// TwinCAT 3 PLC project SAsetGains
// ProgramVersion: 3.1.4023.0
// libraries:
//   Tc2_EtherCAT, * (Beckhoff Automation GmbH)
//   Tc2_Standard, * (Beckhoff Automation GmbH)
//   Tc2_System, * (Beckhoff Automation GmbH)
//   Tc3_Module, * (Beckhoff Automation GmbH)
// project tree:
//   / PlcTask.TcTTO
//   POUs/ clear_fault.TcPOU, MAIN.TcPOU, read_alias.TcPOU, read_dongle.TcPOU, read_ncyl.TcPOU, read_write_SA_gains.TcPOU, save_soc.TcPOU, write_gains.TcPOU
// real-time tasks:
//   TASK PlcTask: cycle T#10ms, priority 20, ADS port 350
// motion (NC):
//   TASK NC-Task 1 SAF: cycle T#2ms, priority 4, ADS port 501
//   TASK NC-Task 1 SVB: cycle T#10ms, priority 8, ADS port 511
//   AXIS Axis 1 (id 1)
//     OtherSettings: AllowMotionCmdToSlave=true
//     encoder EncType=19
//       EncPara: MaxCount=#xffffffff
//     drive DrvType=16
//       DrvPara: MaxCount=#xffffffff, DriveControlDWord=#x00020100
//         Analog: TorqueSetpointScale=10, ScaleFactorActTorque=0.1
//         TimeComp: TaskDelayCycles=1
//     controller CtrType=1
//       CtrPara: PriorControlFactor=1
//         Observer: BandWidth=20
//   AXIS Axis 2 (id 2)
//     OtherSettings: AllowMotionCmdToSlave=true
//     encoder EncType=19
//       EncPara: MaxCount=#xffffffff
//     drive DrvType=16
//       DrvPara: MaxCount=#xffffffff, DriveControlDWord=#x00020100
//         Analog: TorqueSetpointScale=10, ScaleFactorActTorque=0.1
//         TimeComp: TaskDelayCycles=1
//     controller CtrType=1
//       CtrPara: PriorControlFactor=1
//         Observer: BandWidth=20
//   AXIS Axis 3 (id 3)
//     OtherSettings: AllowMotionCmdToSlave=true
//     encoder EncType=19
//       EncPara: MaxCount=#xffffffff
//     drive DrvType=16
//       DrvPara: MaxCount=#xffffffff, DriveControlDWord=#x00020100
//         Analog: TorqueSetpointScale=10, ScaleFactorActTorque=0.1
//         TimeComp: TaskDelayCycles=1
//     controller CtrType=1
//       CtrPara: PriorControlFactor=1
//         Observer: BandWidth=20
//   AXIS Axis 4 (id 4)
//     OtherSettings: AllowMotionCmdToSlave=true
//     encoder EncType=19
//       EncPara: MaxCount=#xffffffff
//     drive DrvType=16
//       DrvPara: MaxCount=#xffffffff, DriveControlDWord=#x00020100
//         Analog: TorqueSetpointScale=10, ScaleFactorActTorque=0.1
//         TimeComp: TaskDelayCycles=1
//     controller CtrType=1
//       CtrPara: PriorControlFactor=1
//         Observer: BandWidth=20
//   AXIS Axis 5 (id 5)
//     OtherSettings: AllowMotionCmdToSlave=true
//     encoder EncType=19
//       EncPara: MaxCount=#xffffffff
//     drive DrvType=16
//       DrvPara: MaxCount=#xffffffff, DriveControlDWord=#x00020100
//         Analog: TorqueSetpointScale=10, ScaleFactorActTorque=0.1
//         TimeComp: TaskDelayCycles=1
//     controller CtrType=1
//       CtrPara: PriorControlFactor=1
//         Observer: BandWidth=20
//   AXIS Axis 6 (id 6)
//     OtherSettings: AllowMotionCmdToSlave=true
//     encoder EncType=19
//       EncPara: MaxCount=#xffffffff
//     drive DrvType=16
//       DrvPara: MaxCount=#xffffffff, DriveControlDWord=#x00020100
//         Analog: TorqueSetpointScale=10, ScaleFactorActTorque=0.1
//         TimeComp: TaskDelayCycles=1
//     controller CtrType=1
//       CtrPara: PriorControlFactor=1
//         Observer: BandWidth=20
// I/O:
//   DEVICE Device 1 (EtherCAT), AmsNetId 10.10.16.19.2.1
//     Box 1 (m1eph) [m1eph]
//       Box 2 (m1sa) [m1sa]
//       Box 3 (m1sa) [m1sa]
//       Box 4 (m1sa) [m1sa]
//       Box 5 (m1sa) [m1sa]
//       Box 6 (m1sa) [m1sa]
//       Box 7 (m1sa) [m1sa]
//       Box 8 (m1sa) [m1sa]
//       Box 9 (m1sa) [m1sa]
//       Box 10 (m1sa) [m1sa]
//       Box 11 (m1sa) [m1sa]
//       Box 12 (m1sa) [m1sa]
//       Box 13 (m1sa) [m1sa]
//       Box 14 (m1sa) [m1sa]
//       Box 15 (m1sa) [m1sa]
//       Box 16 (m1sa) [m1sa]
//       Box 17 (m1sa) [m1sa]
//     Box 18 (m1eph) [m1eph]
//       Box 19 (m1sa) [m1sa]
//       Box 20 (m1sa) [m1sa]
//       Box 21 (m1sa) [m1sa]
//       Box 22 (m1sa) [m1sa]
//       Box 23 (m1sa) [m1sa]
//       Box 24 (m1sa) [m1sa]
//       Box 25 (m1sa) [m1sa]
//       Box 26 (m1sa) [m1sa]
//       Box 27 (m1sa) [m1sa]
//       Box 28 (m1sa) [m1sa]
//       Box 29 (m1sa) [m1sa]
//       Box 30 (m1sa) [m1sa]
//       Box 31 (m1sa) [m1sa]
//       Box 32 (m1sa) [m1sa]
//     Box 33 (m1eph) [m1eph]
//       Box 34 (m1sa) [m1sa]
//       Box 35 (m1sa) [m1sa]
//       Box 36 (m1sa) [m1sa]
//       Box 37 (m1sa) [m1sa]
//       Box 38 (m1sa) [m1sa]
//       Box 39 (m1sa) [m1sa]
//       Box 40 (m1sa) [m1sa]
//       Box 41 (m1sa) [m1sa]
//       Box 42 (m1sa) [m1sa]
//       Box 43 (m1sa) [m1sa]
//       Box 44 (m1sa) [m1sa]
//       Box 45 (m1sa) [m1sa]
//     Box 46 (m1eph) [m1eph]
//       Box 47 (m1sa) [m1sa]
//       Box 48 (m1sa) [m1sa]
//       Box 49 (m1sa) [m1sa]
//       Box 50 (m1sa) [m1sa]
//       Box 51 (m1sa) [m1sa]
//       Box 52 (m1sa) [m1sa]
//       Box 53 (m1sa) [m1sa]
//       Box 54 (m1sa) [m1sa]
//       Box 55 (m1sa) [m1sa]
//       Box 56 (m1sa) [m1sa]
//       Box 57 (m1sa) [m1sa]
//       Box 58 (m1sa) [m1sa]
//       Box 59 (m1sa) [m1sa]
//       Box 60 (m1sa) [m1sa]
//       Box 61 (m1sa) [m1sa]
//       Box 62 (m1sa) [m1sa]
//     Box 63 (m1eph) [m1eph]
//       Box 64 (m1sa) [m1sa]
//       Box 65 (m1sa) [m1sa]
//       Box 66 (m1sa) [m1sa]
//       Box 67 (m1sa) [m1sa]
//       Box 68 (m1sa) [m1sa]
//       Box 69 (m1sa) [m1sa]
//       Box 70 (m1sa) [m1sa]
//       Box 71 (m1sa) [m1sa]
//       Box 72 (m1sa) [m1sa]
//       Box 73 (m1sa) [m1sa]
//       Box 74 (m1sa) [m1sa]
//       Box 75 (m1sa) [m1sa]
//       Box 76 (m1sa) [m1sa]
//       Box 77 (m1sa) [m1sa]
//       Box 78 (m1sa) [m1sa]
//       Box 79 (m1sa) [m1sa]
//     Box 80 (m1eph) [m1eph]
//       Box 81 (m1sa) [m1sa]
//       Box 82 (m1sa) [m1sa]
//       Box 83 (m1sa) [m1sa]
//       Box 84 (m1sa) [m1sa]
//       Box 85 (m1sa) [m1sa]
//       Box 86 (m1sa) [m1sa]
//       Box 87 (m1sa) [m1sa]
//       Box 88 (m1sa) [m1sa]
//       Box 89 (m1sa) [m1sa]
//       Box 90 (m1sa) [m1sa]
//       Box 91 (m1sa) [m1sa]
//       Box 92 (m1sa) [m1sa]
//       Box 93 (m1sa) [m1sa]
//       Box 94 (m1sa) [m1sa]
//       Box 95 (m1sa) [m1sa]
//       Box 96 (m1sa) [m1sa]
//     Box 97 (m1eph) [m1eph]
//       Box 98 (m1sa) [m1sa]
//       Box 99 (m1sa) [m1sa]
//       Box 100 (m1sa) [m1sa]
//       Box 101 (m1sa) [m1sa]
//       Box 102 (m1sa) [m1sa]
//       Box 103 (m1sa) [m1sa]
//       Box 104 (m1sa) [m1sa]
//       Box 105 (m1sa) [m1sa]
//       Box 106 (m1sa) [m1sa]
//       Box 107 (m1sa) [m1sa]
//       Box 108 (m1sa) [m1sa]
//       Box 109 (m1sa) [m1sa]
//       Box 110 (m1sa) [m1sa]
//       Box 111 (m1sa) [m1sa]
//       Box 112 (m1sa) [m1sa]
//       Box 113 (m1sa) [m1sa]
//     Box 114 (m1eph) [m1eph]
//       Box 115 (m1sa) [m1sa]
//       Box 116 (m1sa) [m1sa]
//       Box 117 (m1sa) [m1sa]
//       Box 118 (m1sa) [m1sa]
//       Box 119 (m1sa) [m1sa]
//       Box 120 (m1sa) [m1sa]
//       Box 121 (m1sa) [m1sa]
//       Box 122 (m1sa) [m1sa]
//       Box 123 (m1sa) [m1sa]
//       Box 124 (m1sa) [m1sa]
//       Box 125 (m1sa) [m1sa]
//       Box 126 (m1sa) [m1sa]
//       Box 127 (m1sa) [m1sa]
//       Box 128 (m1sa) [m1sa]
//       Box 129 (m1sa) [m1sa]
//       Box 130 (m1sa) [m1sa]
//     Box 131 (m1eph) [m1eph]
//       Box 132 (m1sa) [m1sa]
//       Box 133 (m1sa) [m1sa]
//       Box 134 (m1sa) [m1sa]
//       Box 135 (m1sa) [m1sa]
//       Box 136 (m1sa) [m1sa]
//       Box 137 (m1sa) [m1sa]
//       Box 138 (m1sa) [m1sa]
//       Box 139 (m1sa) [m1sa]
//       Box 140 (m1sa) [m1sa]
//       Box 141 (m1sa) [m1sa]
//       Box 142 (m1sa) [m1sa]
//       Box 143 (m1sa) [m1sa]
//       Box 144 (m1sa) [m1sa]
//       Box 145 (m1sa) [m1sa]
//       Box 146 (m1sa) [m1sa]
//       Box 147 (m1sa) [m1sa]
//     Box 148 (m1eph) [m1eph]
//       Box 149 (m1sa) [m1sa]
//       Box 150 (m1sa) [m1sa]
//       Box 151 (m1sa) [m1sa]
//       Box 152 (m1sa) [m1sa]
//       Box 153 (m1sa) [m1sa]
//       Box 154 (m1sa) [m1sa]
//       Box 155 (m1sa) [m1sa]
//       Box 156 (m1sa) [m1sa]
//       Box 157 (m1sa) [m1sa]
//       Box 158 (m1sa) [m1sa]
//       Box 159 (m1sa) [m1sa]
//       Box 160 (m1sa) [m1sa]
//       Box 161 (m1sa) [m1sa]
//       Box 162 (m1sa) [m1sa]
//       Box 163 (m1sa) [m1sa]
//       Box 164 (m1sa) [m1sa]
//     Box 165 (m1eph) [m1eph]
//       Box 166 (m1sa) [m1sa]
//       Box 167 (m1sa) [m1sa]
//       Box 168 (m1sa) [m1sa]
//       Box 169 (m1sa) [m1sa]
//       Box 170 (m1sa) [m1sa]
//       Box 171 (m1sa) [m1sa]
//       Box 172 (m1sa) [m1sa]
//       Box 173 (m1sa) [m1sa]
//       Box 174 (m1sa) [m1sa]
//       Box 175 (m1sa) [m1sa]
//       Box 176 (m1sa) [m1sa]
//       Box 177 (m1sa) [m1sa]
//       Box 178 (m1sa) [m1sa]
//       Box 179 (m1sa) [m1sa]
//       Box 180 (m1sa) [m1sa]
//       Box 181 (m1sa) [m1sa]
//     Drive 182 (BEL) [BEL]
//       modules: Module 1 (Cyclic position Mode)
//     Term 183 (EK1100) [EK1100 EtherCAT Coupler (2A E-Bus)]
//       Term 184 (EL5042) [EL5042 2Ch. BiSS-C Encoder]
//       Term 185 (EL3312) [EL3312 2Ch. Ana. Input Thermocouple (TC)]
//       Term 186 (EL9505) [EL9505 Power supply terminal 5V]
//       Term 187 (EL3356-0010) [EL3356-0010 1Ch. Ana. Input Resistor Bridge Terminal, 24bit, High Precision]
//       Term 218 (EL9011) [EL9011 End Terminal]
//     Drive 188 (BEL) [BEL]
//       modules: Module 1 (Cyclic position Mode)
//     Term 189 (EK1100) [EK1100 EtherCAT Coupler (2A E-Bus)]
//       Term 190 (EL5042) [EL5042 2Ch. BiSS-C Encoder]
//       Term 191 (EL3312) [EL3312 2Ch. Ana. Input Thermocouple (TC)]
//       Term 192 (EL9505) [EL9505 Power supply terminal 5V]
//       Term 193 (EL3356-0010) [EL3356-0010 1Ch. Ana. Input Resistor Bridge Terminal, 24bit, High Precision]
//       Term 219 (EL9011) [EL9011 End Terminal]
//     Drive 194 (BEL) [BEL]
//       modules: Module 1 (Cyclic position Mode)
//     Term 195 (EK1100) [EK1100 EtherCAT Coupler (2A E-Bus)]
//       Term 196 (EL5042) [EL5042 2Ch. BiSS-C Encoder]
//       Term 197 (EL3312) [EL3312 2Ch. Ana. Input Thermocouple (TC)]
//       Term 198 (EL9505) [EL9505 Power supply terminal 5V]
//       Term 199 (EL3356-0010) [EL3356-0010 1Ch. Ana. Input Resistor Bridge Terminal, 24bit, High Precision]
//       Term 220 (EL9011) [EL9011 End Terminal]
//     Drive 200 (BEL) [BEL]
//       modules: Module 1 (Cyclic position Mode)
//     Term 201 (EK1100) [EK1100 EtherCAT Coupler (2A E-Bus)]
//       Term 202 (EL5042) [EL5042 2Ch. BiSS-C Encoder]
//       Term 203 (EL3312) [EL3312 2Ch. Ana. Input Thermocouple (TC)]
//       Term 204 (EL9505) [EL9505 Power supply terminal 5V]
//       Term 205 (EL3356-0010) [EL3356-0010 1Ch. Ana. Input Resistor Bridge Terminal, 24bit, High Precision]
//       Term 221 (EL9011) [EL9011 End Terminal]
//     Drive 206 (BEL) [BEL]
//       modules: Module 1 (Cyclic position Mode)
//     Term 207 (EK1100) [EK1100 EtherCAT Coupler (2A E-Bus)]
//       Term 208 (EL5042) [EL5042 2Ch. BiSS-C Encoder]
//       Term 209 (EL3312) [EL3312 2Ch. Ana. Input Thermocouple (TC)]
//       Term 210 (EL9505) [EL9505 Power supply terminal 5V]
//       Term 211 (EL3356-0010) [EL3356-0010 1Ch. Ana. Input Resistor Bridge Terminal, 24bit, High Precision]
//       Term 222 (EL9011) [EL9011 End Terminal]
//     Drive 212 (BEL) [BEL]
//       modules: Module 1 (Cyclic position Mode)
//     Term 213 (EK1100) [EK1100 EtherCAT Coupler (2A E-Bus)]
//       Term 214 (EL5042) [EL5042 2Ch. BiSS-C Encoder]
//       Term 215 (EL3312) [EL3312 2Ch. Ana. Input Thermocouple (TC)]
//       Term 216 (EL9505) [EL9505 Power supply terminal 5V]
//       Term 217 (EL3356-0010) [EL3356-0010 1Ch. Ana. Input Resistor Bridge Terminal, 24bit, High Precision]
//       Term 223 (EL9011) [EL9011 End Terminal]
// variable links:
//   NC-Task 1 SAF/Axes/Axis 1 <-> Device 1 (EtherCAT)/Drive 182 (BEL)
//     Drive/Inputs/In/nDataIn1 <-> Module 1 (Cyclic position Mode)/Cyclic position Inputs/Position loop error
//     Drive/Inputs/In/nDataIn3[0] <-> Module 1 (Cyclic position Mode)/Cyclic position Inputs/Torque actual value
//     Drive/Inputs/In/nDcOutputTime <-> InfoData/DcOutputShift
//     Drive/Inputs/In/nState1 <-> Module 1 (Cyclic position Mode)/Cyclic position Inputs/Status word
//     Drive/Inputs/In/nState2 <-> Module 1 (Cyclic position Mode)/Cyclic position Inputs/Status word @bit 8
//     Drive/Inputs/In/nState4 @bit 1 <-> WcState/InputToggle
//     Drive/Inputs/In/nState4 <-> WcState/WcState
//     Drive/Outputs/Out/nCtrl1 <-> Module 1 (Cyclic position Mode)/Cyclic position Outputs/Control word
//     Drive/Outputs/Out/nCtrl2 <-> Module 1 (Cyclic position Mode)/Cyclic position Outputs/Control word @bit 8
//     Drive/Outputs/Out/nDataOut1 <-> Module 1 (Cyclic position Mode)/Cyclic position Outputs/Profile target position
//     Drive/Outputs/Out/nDataOut3[0] <-> Module 1 (Cyclic position Mode)/Cyclic position Outputs/Torque offset
//     Enc/Inputs/In/nDataIn1 <-> Module 1 (Cyclic position Mode)/Cyclic position Inputs/Actual motor position
//     Enc/Inputs/In/nDataIn7 <-> Module 1 (Cyclic position Mode)/Cyclic position Inputs/Actual motor velocity
//     Enc/Inputs/In/nDcInputTime <-> InfoData/DcInputShift
//     Enc/Inputs/In/nState4 @bit 1 <-> WcState/InputToggle
//     Enc/Inputs/In/nState4 <-> WcState/WcState
//   NC-Task 1 SAF/Axes/Axis 2 <-> Device 1 (EtherCAT)/Drive 188 (BEL)
//     Drive/Inputs/In/nDataIn1 <-> Module 1 (Cyclic position Mode)/Cyclic position Inputs/Position loop error
//     Drive/Inputs/In/nDataIn3[0] <-> Module 1 (Cyclic position Mode)/Cyclic position Inputs/Torque actual value
//     Drive/Inputs/In/nDcOutputTime <-> InfoData/DcOutputShift
//     Drive/Inputs/In/nState1 <-> Module 1 (Cyclic position Mode)/Cyclic position Inputs/Status word
//     Drive/Inputs/In/nState2 <-> Module 1 (Cyclic position Mode)/Cyclic position Inputs/Status word @bit 8
//     Drive/Inputs/In/nState4 @bit 1 <-> WcState/InputToggle
//     Drive/Inputs/In/nState4 <-> WcState/WcState
//     Drive/Outputs/Out/nCtrl1 <-> Module 1 (Cyclic position Mode)/Cyclic position Outputs/Control word
//     Drive/Outputs/Out/nCtrl2 <-> Module 1 (Cyclic position Mode)/Cyclic position Outputs/Control word @bit 8
//     Drive/Outputs/Out/nDataOut1 <-> Module 1 (Cyclic position Mode)/Cyclic position Outputs/Profile target position
//     Drive/Outputs/Out/nDataOut3[0] <-> Module 1 (Cyclic position Mode)/Cyclic position Outputs/Torque offset
//     Enc/Inputs/In/nDataIn1 <-> Module 1 (Cyclic position Mode)/Cyclic position Inputs/Actual motor position
//     Enc/Inputs/In/nDataIn7 <-> Module 1 (Cyclic position Mode)/Cyclic position Inputs/Actual motor velocity
//     Enc/Inputs/In/nDcInputTime <-> InfoData/DcInputShift
//     Enc/Inputs/In/nState4 @bit 1 <-> WcState/InputToggle
//     Enc/Inputs/In/nState4 <-> WcState/WcState
//   NC-Task 1 SAF/Axes/Axis 3 <-> Device 1 (EtherCAT)/Drive 194 (BEL)
//     Drive/Inputs/In/nDataIn1 <-> Module 1 (Cyclic position Mode)/Cyclic position Inputs/Position loop error
//     Drive/Inputs/In/nDataIn3[0] <-> Module 1 (Cyclic position Mode)/Cyclic position Inputs/Torque actual value
//     Drive/Inputs/In/nDcOutputTime <-> InfoData/DcOutputShift
//     Drive/Inputs/In/nState1 <-> Module 1 (Cyclic position Mode)/Cyclic position Inputs/Status word
//     Drive/Inputs/In/nState2 <-> Module 1 (Cyclic position Mode)/Cyclic position Inputs/Status word @bit 8
//     Drive/Inputs/In/nState4 @bit 1 <-> WcState/InputToggle
//     Drive/Inputs/In/nState4 <-> WcState/WcState
//     Drive/Outputs/Out/nCtrl1 <-> Module 1 (Cyclic position Mode)/Cyclic position Outputs/Control word
//     Drive/Outputs/Out/nCtrl2 <-> Module 1 (Cyclic position Mode)/Cyclic position Outputs/Control word @bit 8
//     Drive/Outputs/Out/nDataOut1 <-> Module 1 (Cyclic position Mode)/Cyclic position Outputs/Profile target position
//     Drive/Outputs/Out/nDataOut3[0] <-> Module 1 (Cyclic position Mode)/Cyclic position Outputs/Torque offset
//     Enc/Inputs/In/nDataIn1 <-> Module 1 (Cyclic position Mode)/Cyclic position Inputs/Actual motor position
//     Enc/Inputs/In/nDataIn7 <-> Module 1 (Cyclic position Mode)/Cyclic position Inputs/Actual motor velocity
//     Enc/Inputs/In/nDcInputTime <-> InfoData/DcInputShift
//     Enc/Inputs/In/nState4 @bit 1 <-> WcState/InputToggle
//     Enc/Inputs/In/nState4 <-> WcState/WcState
//   NC-Task 1 SAF/Axes/Axis 4 <-> Device 1 (EtherCAT)/Drive 200 (BEL)
//     Drive/Inputs/In/nDataIn1 <-> Module 1 (Cyclic position Mode)/Cyclic position Inputs/Position loop error
//     Drive/Inputs/In/nDataIn3[0] <-> Module 1 (Cyclic position Mode)/Cyclic position Inputs/Torque actual value
//     Drive/Inputs/In/nDcOutputTime <-> InfoData/DcOutputShift
//     Drive/Inputs/In/nState1 <-> Module 1 (Cyclic position Mode)/Cyclic position Inputs/Status word
//     Drive/Inputs/In/nState2 <-> Module 1 (Cyclic position Mode)/Cyclic position Inputs/Status word @bit 8
//     Drive/Inputs/In/nState4 @bit 1 <-> WcState/InputToggle
//     Drive/Inputs/In/nState4 <-> WcState/WcState
//     Drive/Outputs/Out/nCtrl1 <-> Module 1 (Cyclic position Mode)/Cyclic position Outputs/Control word
//     Drive/Outputs/Out/nCtrl2 <-> Module 1 (Cyclic position Mode)/Cyclic position Outputs/Control word @bit 8
//     Drive/Outputs/Out/nDataOut1 <-> Module 1 (Cyclic position Mode)/Cyclic position Outputs/Profile target position
//     Drive/Outputs/Out/nDataOut3[0] <-> Module 1 (Cyclic position Mode)/Cyclic position Outputs/Torque offset
//     Enc/Inputs/In/nDataIn1 <-> Module 1 (Cyclic position Mode)/Cyclic position Inputs/Actual motor position
//     Enc/Inputs/In/nDataIn7 <-> Module 1 (Cyclic position Mode)/Cyclic position Inputs/Actual motor velocity
//     Enc/Inputs/In/nDcInputTime <-> InfoData/DcInputShift
//     Enc/Inputs/In/nState4 @bit 1 <-> WcState/InputToggle
//     Enc/Inputs/In/nState4 <-> WcState/WcState
//   NC-Task 1 SAF/Axes/Axis 5 <-> Device 1 (EtherCAT)/Drive 206 (BEL)
//     Drive/Inputs/In/nDataIn1 <-> Module 1 (Cyclic position Mode)/Cyclic position Inputs/Position loop error
//     Drive/Inputs/In/nDataIn3[0] <-> Module 1 (Cyclic position Mode)/Cyclic position Inputs/Torque actual value
//     Drive/Inputs/In/nDcOutputTime <-> InfoData/DcOutputShift
//     Drive/Inputs/In/nState1 <-> Module 1 (Cyclic position Mode)/Cyclic position Inputs/Status word
//     Drive/Inputs/In/nState2 <-> Module 1 (Cyclic position Mode)/Cyclic position Inputs/Status word @bit 8
//     Drive/Inputs/In/nState4 @bit 1 <-> WcState/InputToggle
//     Drive/Inputs/In/nState4 <-> WcState/WcState
//     Drive/Outputs/Out/nCtrl1 <-> Module 1 (Cyclic position Mode)/Cyclic position Outputs/Control word
//     Drive/Outputs/Out/nCtrl2 <-> Module 1 (Cyclic position Mode)/Cyclic position Outputs/Control word @bit 8
//     Drive/Outputs/Out/nDataOut1 <-> Module 1 (Cyclic position Mode)/Cyclic position Outputs/Profile target position
//     Drive/Outputs/Out/nDataOut3[0] <-> Module 1 (Cyclic position Mode)/Cyclic position Outputs/Torque offset
//     Enc/Inputs/In/nDataIn1 <-> Module 1 (Cyclic position Mode)/Cyclic position Inputs/Actual motor position
//     Enc/Inputs/In/nDataIn7 <-> Module 1 (Cyclic position Mode)/Cyclic position Inputs/Actual motor velocity
//     Enc/Inputs/In/nDcInputTime <-> InfoData/DcInputShift
//     Enc/Inputs/In/nState4 @bit 1 <-> WcState/InputToggle
//     Enc/Inputs/In/nState4 <-> WcState/WcState
//   NC-Task 1 SAF/Axes/Axis 6 <-> Device 1 (EtherCAT)/Drive 212 (BEL)
//     Drive/Inputs/In/nDataIn1 <-> Module 1 (Cyclic position Mode)/Cyclic position Inputs/Position loop error
//     Drive/Inputs/In/nDataIn3[0] <-> Module 1 (Cyclic position Mode)/Cyclic position Inputs/Torque actual value
//     Drive/Inputs/In/nDcOutputTime <-> InfoData/DcOutputShift
//     Drive/Inputs/In/nState1 <-> Module 1 (Cyclic position Mode)/Cyclic position Inputs/Status word
//     Drive/Inputs/In/nState2 <-> Module 1 (Cyclic position Mode)/Cyclic position Inputs/Status word @bit 8
//     Drive/Inputs/In/nState4 @bit 1 <-> WcState/InputToggle
//     Drive/Inputs/In/nState4 <-> WcState/WcState
//     Drive/Outputs/Out/nCtrl1 <-> Module 1 (Cyclic position Mode)/Cyclic position Outputs/Control word
//     Drive/Outputs/Out/nCtrl2 <-> Module 1 (Cyclic position Mode)/Cyclic position Outputs/Control word @bit 8
//     Drive/Outputs/Out/nDataOut1 <-> Module 1 (Cyclic position Mode)/Cyclic position Outputs/Profile target position
//     Drive/Outputs/Out/nDataOut3[0] <-> Module 1 (Cyclic position Mode)/Cyclic position Outputs/Torque offset
//     Enc/Inputs/In/nDataIn1 <-> Module 1 (Cyclic position Mode)/Cyclic position Inputs/Actual motor position
//     Enc/Inputs/In/nDataIn7 <-> Module 1 (Cyclic position Mode)/Cyclic position Inputs/Actual motor velocity
//     Enc/Inputs/In/nDcInputTime <-> InfoData/DcInputShift
//     Enc/Inputs/In/nState4 @bit 1 <-> WcState/InputToggle
//     Enc/Inputs/In/nState4 <-> WcState/WcState
//   SAsetGains/SAsetGains Instance <-> Device 1 (EtherCAT)
//     PlcTask Inputs/MAIN.FrmWcStat[1] <-> Inputs/Frm0WcState
//   SAsetGains/SAsetGains Instance <-> Device 1 (EtherCAT)/Box 1 (m1eph)
//     PlcTask Outputs/MAIN.msthb[1] <-> Control process data mapping/msthb
//   SAsetGains/SAsetGains Instance <-> Device 1 (EtherCAT)/Box 1 (m1eph)/Box 10 (m1sa)
//     PlcTask Inputs/MAIN.cloop_stat[9] <-> Status process data mapping/close_loop
//     PlcTask Inputs/MAIN.enable_stat[9] <-> Status process data mapping/enable
//     PlcTask Inputs/MAIN.force_rb_X[9] <-> Status process data mapping/force_rb_X
//     PlcTask Inputs/MAIN.force_rb_Y[9] <-> Status process data mapping/force_rb_Y
//     PlcTask Inputs/MAIN.force_rb_Z[9] <-> Status process data mapping/force_rb_Z
//     PlcTask Inputs/MAIN.force_sp_X[9] <-> Status process data mapping/force_sp_X
//     PlcTask Inputs/MAIN.force_sp_Y[9] <-> Status process data mapping/force_sp_Y
//     PlcTask Inputs/MAIN.force_sp_Z[9] <-> Status process data mapping/force_sp_Z
//     PlcTask Inputs/MAIN.pwm1[9] <-> Status process data mapping/pwm1
//     PlcTask Inputs/MAIN.pwm2[9] <-> Status process data mapping/pwm2
//     PlcTask Inputs/MAIN.pwm3[9] <-> Status process data mapping/pwm3
//     PlcTask Outputs/MAIN.enable_cmd[9] <-> Control process data mapping/enable
//     PlcTask Outputs/MAIN.force_cmd_X[9] <-> Control process data mapping/force_sp_X
//     PlcTask Outputs/MAIN.force_cmd_Y[9] <-> Control process data mapping/force_sp_Y
//     PlcTask Outputs/MAIN.force_cmd_Z[9] <-> Control process data mapping/force_sp_Z
//     PlcTask Outputs/MAIN.msthb[10] <-> Control process data mapping/msthb
//   SAsetGains/SAsetGains Instance <-> Device 1 (EtherCAT)/Box 1 (m1eph)/Box 11 (m1sa)
//     PlcTask Inputs/MAIN.cloop_stat[10] <-> Status process data mapping/close_loop
//     PlcTask Inputs/MAIN.enable_stat[10] <-> Status process data mapping/enable
//     PlcTask Inputs/MAIN.force_rb_X[10] <-> Status process data mapping/force_rb_X
//     PlcTask Inputs/MAIN.force_rb_Y[10] <-> Status process data mapping/force_rb_Y
//     PlcTask Inputs/MAIN.force_rb_Z[10] <-> Status process data mapping/force_rb_Z
//     PlcTask Inputs/MAIN.force_sp_X[10] <-> Status process data mapping/force_sp_X
//     PlcTask Inputs/MAIN.force_sp_Y[10] <-> Status process data mapping/force_sp_Y
//     PlcTask Inputs/MAIN.force_sp_Z[10] <-> Status process data mapping/force_sp_Z
//     PlcTask Inputs/MAIN.pwm1[10] <-> Status process data mapping/pwm1
//     PlcTask Inputs/MAIN.pwm2[10] <-> Status process data mapping/pwm2
//     PlcTask Inputs/MAIN.pwm3[10] <-> Status process data mapping/pwm3
//     PlcTask Outputs/MAIN.enable_cmd[10] <-> Control process data mapping/enable
//     PlcTask Outputs/MAIN.force_cmd_X[10] <-> Control process data mapping/force_sp_X
//     PlcTask Outputs/MAIN.force_cmd_Y[10] <-> Control process data mapping/force_sp_Y
//     PlcTask Outputs/MAIN.force_cmd_Z[10] <-> Control process data mapping/force_sp_Z
//     PlcTask Outputs/MAIN.msthb[11] <-> Control process data mapping/msthb
//   SAsetGains/SAsetGains Instance <-> Device 1 (EtherCAT)/Box 1 (m1eph)/Box 12 (m1sa)
//     PlcTask Inputs/MAIN.cloop_stat[11] <-> Status process data mapping/close_loop
//     PlcTask Inputs/MAIN.enable_stat[11] <-> Status process data mapping/enable
//     PlcTask Inputs/MAIN.force_rb_X[11] <-> Status process data mapping/force_rb_X
//     PlcTask Inputs/MAIN.force_rb_Y[11] <-> Status process data mapping/force_rb_Y
//     PlcTask Inputs/MAIN.force_rb_Z[11] <-> Status process data mapping/force_rb_Z
//     PlcTask Inputs/MAIN.force_sp_X[11] <-> Status process data mapping/force_sp_X
//     PlcTask Inputs/MAIN.force_sp_Y[11] <-> Status process data mapping/force_sp_Y
//     PlcTask Inputs/MAIN.force_sp_Z[11] <-> Status process data mapping/force_sp_Z
//     PlcTask Inputs/MAIN.pwm1[11] <-> Status process data mapping/pwm1
//     PlcTask Inputs/MAIN.pwm2[11] <-> Status process data mapping/pwm2
//     PlcTask Inputs/MAIN.pwm3[11] <-> Status process data mapping/pwm3
//     PlcTask Outputs/MAIN.enable_cmd[11] <-> Control process data mapping/enable
//     PlcTask Outputs/MAIN.force_cmd_X[11] <-> Control process data mapping/force_sp_X
//     PlcTask Outputs/MAIN.force_cmd_Y[11] <-> Control process data mapping/force_sp_Y
//     PlcTask Outputs/MAIN.force_cmd_Z[11] <-> Control process data mapping/force_sp_Z
//     PlcTask Outputs/MAIN.msthb[12] <-> Control process data mapping/msthb
//   SAsetGains/SAsetGains Instance <-> Device 1 (EtherCAT)/Box 1 (m1eph)/Box 13 (m1sa)
//     PlcTask Inputs/MAIN.cloop_stat[12] <-> Status process data mapping/close_loop
//     PlcTask Inputs/MAIN.enable_stat[12] <-> Status process data mapping/enable
//     PlcTask Inputs/MAIN.force_rb_X[12] <-> Status process data mapping/force_rb_X
//     PlcTask Inputs/MAIN.force_rb_Y[12] <-> Status process data mapping/force_rb_Y
//     PlcTask Inputs/MAIN.force_rb_Z[12] <-> Status process data mapping/force_rb_Z
//     PlcTask Inputs/MAIN.force_sp_X[12] <-> Status process data mapping/force_sp_X
//     PlcTask Inputs/MAIN.force_sp_Y[12] <-> Status process data mapping/force_sp_Y
//     PlcTask Inputs/MAIN.force_sp_Z[12] <-> Status process data mapping/force_sp_Z
//     PlcTask Inputs/MAIN.pwm1[12] <-> Status process data mapping/pwm1
//     PlcTask Inputs/MAIN.pwm2[12] <-> Status process data mapping/pwm2
//     PlcTask Inputs/MAIN.pwm3[12] <-> Status process data mapping/pwm3
//     PlcTask Outputs/MAIN.enable_cmd[12] <-> Control process data mapping/enable
//     PlcTask Outputs/MAIN.force_cmd_X[12] <-> Control process data mapping/force_sp_X
//     PlcTask Outputs/MAIN.force_cmd_Y[12] <-> Control process data mapping/force_sp_Y
//     PlcTask Outputs/MAIN.force_cmd_Z[12] <-> Control process data mapping/force_sp_Z
//     PlcTask Outputs/MAIN.msthb[13] <-> Control process data mapping/msthb
//   SAsetGains/SAsetGains Instance <-> Device 1 (EtherCAT)/Box 1 (m1eph)/Box 14 (m1sa)
//     PlcTask Inputs/MAIN.cloop_stat[13] <-> Status process data mapping/close_loop
//     PlcTask Inputs/MAIN.enable_stat[13] <-> Status process data mapping/enable
//     PlcTask Inputs/MAIN.force_rb_X[13] <-> Status process data mapping/force_rb_X
//     PlcTask Inputs/MAIN.force_rb_Y[13] <-> Status process data mapping/force_rb_Y
//     PlcTask Inputs/MAIN.force_rb_Z[13] <-> Status process data mapping/force_rb_Z
//     PlcTask Inputs/MAIN.force_sp_X[13] <-> Status process data mapping/force_sp_X
//     PlcTask Inputs/MAIN.force_sp_Y[13] <-> Status process data mapping/force_sp_Y
//     PlcTask Inputs/MAIN.force_sp_Z[13] <-> Status process data mapping/force_sp_Z
//     PlcTask Inputs/MAIN.pwm1[13] <-> Status process data mapping/pwm1
//     PlcTask Inputs/MAIN.pwm2[13] <-> Status process data mapping/pwm2
//     PlcTask Inputs/MAIN.pwm3[13] <-> Status process data mapping/pwm3
//     PlcTask Outputs/MAIN.enable_cmd[13] <-> Control process data mapping/enable
//     PlcTask Outputs/MAIN.force_cmd_X[13] <-> Control process data mapping/force_sp_X
//     PlcTask Outputs/MAIN.force_cmd_Y[13] <-> Control process data mapping/force_sp_Y
//     PlcTask Outputs/MAIN.force_cmd_Z[13] <-> Control process data mapping/force_sp_Z
//     PlcTask Outputs/MAIN.msthb[14] <-> Control process data mapping/msthb
//   SAsetGains/SAsetGains Instance <-> Device 1 (EtherCAT)/Box 1 (m1eph)/Box 15 (m1sa)
//     PlcTask Inputs/MAIN.cloop_stat[14] <-> Status process data mapping/close_loop
//     PlcTask Inputs/MAIN.enable_stat[14] <-> Status process data mapping/enable
//     PlcTask Inputs/MAIN.force_rb_X[14] <-> Status process data mapping/force_rb_X
//     PlcTask Inputs/MAIN.force_rb_Y[14] <-> Status process data mapping/force_rb_Y
//     PlcTask Inputs/MAIN.force_rb_Z[14] <-> Status process data mapping/force_rb_Z
//     PlcTask Inputs/MAIN.force_sp_X[14] <-> Status process data mapping/force_sp_X
//     PlcTask Inputs/MAIN.force_sp_Y[14] <-> Status process data mapping/force_sp_Y
//     PlcTask Inputs/MAIN.force_sp_Z[14] <-> Status process data mapping/force_sp_Z
//     PlcTask Inputs/MAIN.pwm1[14] <-> Status process data mapping/pwm1
//     PlcTask Inputs/MAIN.pwm2[14] <-> Status process data mapping/pwm2
//     PlcTask Inputs/MAIN.pwm3[14] <-> Status process data mapping/pwm3
//     PlcTask Outputs/MAIN.enable_cmd[14] <-> Control process data mapping/enable
//     PlcTask Outputs/MAIN.force_cmd_X[14] <-> Control process data mapping/force_sp_X
//     PlcTask Outputs/MAIN.force_cmd_Y[14] <-> Control process data mapping/force_sp_Y
//     PlcTask Outputs/MAIN.force_cmd_Z[14] <-> Control process data mapping/force_sp_Z
//     PlcTask Outputs/MAIN.msthb[15] <-> Control process data mapping/msthb
//   SAsetGains/SAsetGains Instance <-> Device 1 (EtherCAT)/Box 1 (m1eph)/Box 16 (m1sa)
//     PlcTask Inputs/MAIN.cloop_stat[15] <-> Status process data mapping/close_loop
//     PlcTask Inputs/MAIN.enable_stat[15] <-> Status process data mapping/enable
//     PlcTask Inputs/MAIN.force_rb_X[15] <-> Status process data mapping/force_rb_X
//     PlcTask Inputs/MAIN.force_rb_Y[15] <-> Status process data mapping/force_rb_Y
//     PlcTask Inputs/MAIN.force_rb_Z[15] <-> Status process data mapping/force_rb_Z
//     PlcTask Inputs/MAIN.force_sp_X[15] <-> Status process data mapping/force_sp_X
//     PlcTask Inputs/MAIN.force_sp_Y[15] <-> Status process data mapping/force_sp_Y
//     PlcTask Inputs/MAIN.force_sp_Z[15] <-> Status process data mapping/force_sp_Z
//     PlcTask Inputs/MAIN.pwm1[15] <-> Status process data mapping/pwm1
//     PlcTask Inputs/MAIN.pwm2[15] <-> Status process data mapping/pwm2
//     PlcTask Inputs/MAIN.pwm3[15] <-> Status process data mapping/pwm3
//     PlcTask Outputs/MAIN.enable_cmd[15] <-> Control process data mapping/enable
//     PlcTask Outputs/MAIN.force_cmd_X[15] <-> Control process data mapping/force_sp_X
//     PlcTask Outputs/MAIN.force_cmd_Y[15] <-> Control process data mapping/force_sp_Y
//     PlcTask Outputs/MAIN.force_cmd_Z[15] <-> Control process data mapping/force_sp_Z
//     PlcTask Outputs/MAIN.msthb[16] <-> Control process data mapping/msthb
//   SAsetGains/SAsetGains Instance <-> Device 1 (EtherCAT)/Box 1 (m1eph)/Box 17 (m1sa)
//     PlcTask Inputs/MAIN.cloop_stat[16] <-> Status process data mapping/close_loop
//     PlcTask Inputs/MAIN.enable_stat[16] <-> Status process data mapping/enable
//     PlcTask Inputs/MAIN.force_rb_X[16] <-> Status process data mapping/force_rb_X
//     PlcTask Inputs/MAIN.force_rb_Y[16] <-> Status process data mapping/force_rb_Y
//     PlcTask Inputs/MAIN.force_rb_Z[16] <-> Status process data mapping/force_rb_Z
//     PlcTask Inputs/MAIN.force_sp_X[16] <-> Status process data mapping/force_sp_X
//     PlcTask Inputs/MAIN.force_sp_Y[16] <-> Status process data mapping/force_sp_Y
//     PlcTask Inputs/MAIN.force_sp_Z[16] <-> Status process data mapping/force_sp_Z
//     PlcTask Inputs/MAIN.pwm1[16] <-> Status process data mapping/pwm1
//     PlcTask Inputs/MAIN.pwm2[16] <-> Status process data mapping/pwm2
//     PlcTask Inputs/MAIN.pwm3[16] <-> Status process data mapping/pwm3
//     PlcTask Outputs/MAIN.enable_cmd[16] <-> Control process data mapping/enable
//     PlcTask Outputs/MAIN.force_cmd_X[16] <-> Control process data mapping/force_sp_X
//     PlcTask Outputs/MAIN.force_cmd_Y[16] <-> Control process data mapping/force_sp_Y
//     PlcTask Outputs/MAIN.force_cmd_Z[16] <-> Control process data mapping/force_sp_Z
//     PlcTask Outputs/MAIN.msthb[17] <-> Control process data mapping/msthb
//   SAsetGains/SAsetGains Instance <-> Device 1 (EtherCAT)/Box 1 (m1eph)/Box 2 (m1sa)
//     PlcTask Inputs/MAIN.cloop_stat[1] <-> Status process data mapping/close_loop
//     PlcTask Inputs/MAIN.enable_stat[1] <-> Status process data mapping/enable
//     PlcTask Inputs/MAIN.force_rb_X[1] <-> Status process data mapping/force_rb_X
//     PlcTask Inputs/MAIN.force_rb_Y[1] <-> Status process data mapping/force_rb_Y
//     PlcTask Inputs/MAIN.force_rb_Z[1] <-> Status process data mapping/force_rb_Z
//     PlcTask Inputs/MAIN.force_sp_X[1] <-> Status process data mapping/force_sp_X
//     PlcTask Inputs/MAIN.force_sp_Y[1] <-> Status process data mapping/force_sp_Y
//     PlcTask Inputs/MAIN.force_sp_Z[1] <-> Status process data mapping/force_sp_Z
//     PlcTask Inputs/MAIN.pwm1[1] <-> Status process data mapping/pwm1
//     PlcTask Inputs/MAIN.pwm2[1] <-> Status process data mapping/pwm2
//     PlcTask Inputs/MAIN.pwm3[1] <-> Status process data mapping/pwm3
//     PlcTask Outputs/MAIN.enable_cmd[1] <-> Control process data mapping/enable
//     PlcTask Outputs/MAIN.force_cmd_X[1] <-> Control process data mapping/force_sp_X
//     PlcTask Outputs/MAIN.force_cmd_Y[1] <-> Control process data mapping/force_sp_Y
//     PlcTask Outputs/MAIN.force_cmd_Z[1] <-> Control process data mapping/force_sp_Z
//     PlcTask Outputs/MAIN.msthb[2] <-> Control process data mapping/msthb
//   SAsetGains/SAsetGains Instance <-> Device 1 (EtherCAT)/Box 1 (m1eph)/Box 3 (m1sa)
//     PlcTask Inputs/MAIN.cloop_stat[2] <-> Status process data mapping/close_loop
//     PlcTask Inputs/MAIN.enable_stat[2] <-> Status process data mapping/enable
//     PlcTask Inputs/MAIN.force_rb_X[2] <-> Status process data mapping/force_rb_X
//     PlcTask Inputs/MAIN.force_rb_Y[2] <-> Status process data mapping/force_rb_Y
//     PlcTask Inputs/MAIN.force_rb_Z[2] <-> Status process data mapping/force_rb_Z
//     PlcTask Inputs/MAIN.force_sp_X[2] <-> Status process data mapping/force_sp_X
//     PlcTask Inputs/MAIN.force_sp_Y[2] <-> Status process data mapping/force_sp_Y
//     PlcTask Inputs/MAIN.force_sp_Z[2] <-> Status process data mapping/force_sp_Z
//     PlcTask Inputs/MAIN.pwm1[2] <-> Status process data mapping/pwm1
//     PlcTask Inputs/MAIN.pwm2[2] <-> Status process data mapping/pwm2
//     PlcTask Inputs/MAIN.pwm3[2] <-> Status process data mapping/pwm3
//     PlcTask Outputs/MAIN.enable_cmd[2] <-> Control process data mapping/enable
//     PlcTask Outputs/MAIN.force_cmd_X[2] <-> Control process data mapping/force_sp_X
//     PlcTask Outputs/MAIN.force_cmd_Y[2] <-> Control process data mapping/force_sp_Y
//     PlcTask Outputs/MAIN.force_cmd_Z[2] <-> Control process data mapping/force_sp_Z
//     PlcTask Outputs/MAIN.msthb[3] <-> Control process data mapping/msthb
//   SAsetGains/SAsetGains Instance <-> Device 1 (EtherCAT)/Box 1 (m1eph)/Box 4 (m1sa)
//     PlcTask Inputs/MAIN.cloop_stat[3] <-> Status process data mapping/close_loop
//     PlcTask Inputs/MAIN.enable_stat[3] <-> Status process data mapping/enable
//     PlcTask Inputs/MAIN.force_rb_X[3] <-> Status process data mapping/force_rb_X
//     PlcTask Inputs/MAIN.force_rb_Y[3] <-> Status process data mapping/force_rb_Y
//     PlcTask Inputs/MAIN.force_rb_Z[3] <-> Status process data mapping/force_rb_Z
//     PlcTask Inputs/MAIN.force_sp_X[3] <-> Status process data mapping/force_sp_X
//     PlcTask Inputs/MAIN.force_sp_Y[3] <-> Status process data mapping/force_sp_Y
//     PlcTask Inputs/MAIN.force_sp_Z[3] <-> Status process data mapping/force_sp_Z
//     PlcTask Inputs/MAIN.pwm1[3] <-> Status process data mapping/pwm1
//     PlcTask Inputs/MAIN.pwm2[3] <-> Status process data mapping/pwm2
//     PlcTask Inputs/MAIN.pwm3[3] <-> Status process data mapping/pwm3
//     PlcTask Outputs/MAIN.enable_cmd[3] <-> Control process data mapping/enable
//     PlcTask Outputs/MAIN.force_cmd_X[3] <-> Control process data mapping/force_sp_X
//     PlcTask Outputs/MAIN.force_cmd_Y[3] <-> Control process data mapping/force_sp_Y
//     PlcTask Outputs/MAIN.force_cmd_Z[3] <-> Control process data mapping/force_sp_Z
//     PlcTask Outputs/MAIN.msthb[4] <-> Control process data mapping/msthb
//   SAsetGains/SAsetGains Instance <-> Device 1 (EtherCAT)/Box 1 (m1eph)/Box 5 (m1sa)
//     PlcTask Inputs/MAIN.cloop_stat[4] <-> Status process data mapping/close_loop
//     PlcTask Inputs/MAIN.enable_stat[4] <-> Status process data mapping/enable
//     PlcTask Inputs/MAIN.force_rb_X[4] <-> Status process data mapping/force_rb_X
//     PlcTask Inputs/MAIN.force_rb_Y[4] <-> Status process data mapping/force_rb_Y
//     PlcTask Inputs/MAIN.force_rb_Z[4] <-> Status process data mapping/force_rb_Z
//     PlcTask Inputs/MAIN.force_sp_X[4] <-> Status process data mapping/force_sp_X
//     PlcTask Inputs/MAIN.force_sp_Y[4] <-> Status process data mapping/force_sp_Y
//     PlcTask Inputs/MAIN.force_sp_Z[4] <-> Status process data mapping/force_sp_Z
//     PlcTask Inputs/MAIN.pwm1[4] <-> Status process data mapping/pwm1
//     PlcTask Inputs/MAIN.pwm2[4] <-> Status process data mapping/pwm2
//     PlcTask Inputs/MAIN.pwm3[4] <-> Status process data mapping/pwm3
//     PlcTask Outputs/MAIN.enable_cmd[4] <-> Control process data mapping/enable
//     PlcTask Outputs/MAIN.force_cmd_X[4] <-> Control process data mapping/force_sp_X
//     PlcTask Outputs/MAIN.force_cmd_Y[4] <-> Control process data mapping/force_sp_Y
//     PlcTask Outputs/MAIN.force_cmd_Z[4] <-> Control process data mapping/force_sp_Z
//     PlcTask Outputs/MAIN.msthb[5] <-> Control process data mapping/msthb
//   SAsetGains/SAsetGains Instance <-> Device 1 (EtherCAT)/Box 1 (m1eph)/Box 6 (m1sa)
//     PlcTask Inputs/MAIN.cloop_stat[5] <-> Status process data mapping/close_loop
//     PlcTask Inputs/MAIN.enable_stat[5] <-> Status process data mapping/enable
//     PlcTask Inputs/MAIN.force_rb_X[5] <-> Status process data mapping/force_rb_X
//     PlcTask Inputs/MAIN.force_rb_Y[5] <-> Status process data mapping/force_rb_Y
//     PlcTask Inputs/MAIN.force_rb_Z[5] <-> Status process data mapping/force_rb_Z
//     PlcTask Inputs/MAIN.force_sp_X[5] <-> Status process data mapping/force_sp_X
//     PlcTask Inputs/MAIN.force_sp_Y[5] <-> Status process data mapping/force_sp_Y
//     PlcTask Inputs/MAIN.force_sp_Z[5] <-> Status process data mapping/force_sp_Z
//     PlcTask Inputs/MAIN.pwm1[5] <-> Status process data mapping/pwm1
//     PlcTask Inputs/MAIN.pwm2[5] <-> Status process data mapping/pwm2
//     PlcTask Inputs/MAIN.pwm3[5] <-> Status process data mapping/pwm3
//     PlcTask Outputs/MAIN.enable_cmd[5] <-> Control process data mapping/enable
//     PlcTask Outputs/MAIN.force_cmd_X[5] <-> Control process data mapping/force_sp_X
//     PlcTask Outputs/MAIN.force_cmd_Y[5] <-> Control process data mapping/force_sp_Y
//     PlcTask Outputs/MAIN.force_cmd_Z[5] <-> Control process data mapping/force_sp_Z
//     PlcTask Outputs/MAIN.msthb[6] <-> Control process data mapping/msthb
//   SAsetGains/SAsetGains Instance <-> Device 1 (EtherCAT)/Box 1 (m1eph)/Box 7 (m1sa)
//     PlcTask Inputs/MAIN.cloop_stat[6] <-> Status process data mapping/close_loop
//     PlcTask Inputs/MAIN.enable_stat[6] <-> Status process data mapping/enable
//     PlcTask Inputs/MAIN.force_rb_X[6] <-> Status process data mapping/force_rb_X
//     PlcTask Inputs/MAIN.force_rb_Y[6] <-> Status process data mapping/force_rb_Y
//     PlcTask Inputs/MAIN.force_rb_Z[6] <-> Status process data mapping/force_rb_Z
//     PlcTask Inputs/MAIN.force_sp_X[6] <-> Status process data mapping/force_sp_X
//     PlcTask Inputs/MAIN.force_sp_Y[6] <-> Status process data mapping/force_sp_Y
//     PlcTask Inputs/MAIN.force_sp_Z[6] <-> Status process data mapping/force_sp_Z
//     PlcTask Inputs/MAIN.pwm1[6] <-> Status process data mapping/pwm1
//     PlcTask Inputs/MAIN.pwm2[6] <-> Status process data mapping/pwm2
//     PlcTask Inputs/MAIN.pwm3[6] <-> Status process data mapping/pwm3
//     PlcTask Outputs/MAIN.enable_cmd[6] <-> Control process data mapping/enable
//     PlcTask Outputs/MAIN.force_cmd_X[6] <-> Control process data mapping/force_sp_X
//     PlcTask Outputs/MAIN.force_cmd_Y[6] <-> Control process data mapping/force_sp_Y
//     PlcTask Outputs/MAIN.force_cmd_Z[6] <-> Control process data mapping/force_sp_Z
//     PlcTask Outputs/MAIN.msthb[7] <-> Control process data mapping/msthb
//   SAsetGains/SAsetGains Instance <-> Device 1 (EtherCAT)/Box 1 (m1eph)/Box 8 (m1sa)
//     PlcTask Inputs/MAIN.cloop_stat[7] <-> Status process data mapping/close_loop
//     PlcTask Inputs/MAIN.enable_stat[7] <-> Status process data mapping/enable
//     PlcTask Inputs/MAIN.force_rb_X[7] <-> Status process data mapping/force_rb_X
//     PlcTask Inputs/MAIN.force_rb_Y[7] <-> Status process data mapping/force_rb_Y
//     PlcTask Inputs/MAIN.force_rb_Z[7] <-> Status process data mapping/force_rb_Z
//     PlcTask Inputs/MAIN.force_sp_X[7] <-> Status process data mapping/force_sp_X
//     PlcTask Inputs/MAIN.force_sp_Y[7] <-> Status process data mapping/force_sp_Y
//     PlcTask Inputs/MAIN.force_sp_Z[7] <-> Status process data mapping/force_sp_Z
//     PlcTask Inputs/MAIN.pwm1[7] <-> Status process data mapping/pwm1
//     PlcTask Inputs/MAIN.pwm2[7] <-> Status process data mapping/pwm2
//     PlcTask Inputs/MAIN.pwm3[7] <-> Status process data mapping/pwm3
//     PlcTask Outputs/MAIN.enable_cmd[7] <-> Control process data mapping/enable
//     PlcTask Outputs/MAIN.force_cmd_X[7] <-> Control process data mapping/force_sp_X
//     PlcTask Outputs/MAIN.force_cmd_Y[7] <-> Control process data mapping/force_sp_Y
//     PlcTask Outputs/MAIN.force_cmd_Z[7] <-> Control process data mapping/force_sp_Z
//     PlcTask Outputs/MAIN.msthb[8] <-> Control process data mapping/msthb
//   SAsetGains/SAsetGains Instance <-> Device 1 (EtherCAT)/Box 1 (m1eph)/Box 9 (m1sa)
//     PlcTask Inputs/MAIN.cloop_stat[8] <-> Status process data mapping/close_loop
//     PlcTask Inputs/MAIN.enable_stat[8] <-> Status process data mapping/enable
//     PlcTask Inputs/MAIN.force_rb_X[8] <-> Status process data mapping/force_rb_X
//     PlcTask Inputs/MAIN.force_rb_Y[8] <-> Status process data mapping/force_rb_Y
//     PlcTask Inputs/MAIN.force_rb_Z[8] <-> Status process data mapping/force_rb_Z
//     PlcTask Inputs/MAIN.force_sp_X[8] <-> Status process data mapping/force_sp_X
//     PlcTask Inputs/MAIN.force_sp_Y[8] <-> Status process data mapping/force_sp_Y
//     PlcTask Inputs/MAIN.force_sp_Z[8] <-> Status process data mapping/force_sp_Z
//     PlcTask Inputs/MAIN.pwm1[8] <-> Status process data mapping/pwm1
//     PlcTask Inputs/MAIN.pwm2[8] <-> Status process data mapping/pwm2
//     PlcTask Inputs/MAIN.pwm3[8] <-> Status process data mapping/pwm3
//     PlcTask Outputs/MAIN.enable_cmd[8] <-> Control process data mapping/enable
//     PlcTask Outputs/MAIN.force_cmd_X[8] <-> Control process data mapping/force_sp_X
//     PlcTask Outputs/MAIN.force_cmd_Y[8] <-> Control process data mapping/force_sp_Y
//     PlcTask Outputs/MAIN.force_cmd_Z[8] <-> Control process data mapping/force_sp_Z
//     PlcTask Outputs/MAIN.msthb[9] <-> Control process data mapping/msthb
//   SAsetGains/SAsetGains Instance <-> Device 1 (EtherCAT)/Box 114 (m1eph)
//     PlcTask Outputs/MAIN.msthb[114] <-> Control process data mapping/msthb
//   SAsetGains/SAsetGains Instance <-> Device 1 (EtherCAT)/Box 114 (m1eph)/Box 115 (m1sa)
//     PlcTask Inputs/MAIN.cloop_stat[107] <-> Status process data mapping/close_loop
//     PlcTask Inputs/MAIN.enable_stat[107] <-> Status process data mapping/enable
//     PlcTask Inputs/MAIN.force_rb_X[107] <-> Status process data mapping/force_rb_X
//     PlcTask Inputs/MAIN.force_rb_Y[107] <-> Status process data mapping/force_rb_Y
//     PlcTask Inputs/MAIN.force_rb_Z[107] <-> Status process data mapping/force_rb_Z
//     PlcTask Inputs/MAIN.force_sp_X[107] <-> Status process data mapping/force_sp_X
//     PlcTask Inputs/MAIN.force_sp_Y[107] <-> Status process data mapping/force_sp_Y
//     PlcTask Inputs/MAIN.force_sp_Z[107] <-> Status process data mapping/force_sp_Z
//     PlcTask Inputs/MAIN.pwm1[107] <-> Status process data mapping/pwm1
//     PlcTask Inputs/MAIN.pwm2[107] <-> Status process data mapping/pwm2
//     PlcTask Inputs/MAIN.pwm3[107] <-> Status process data mapping/pwm3
//     PlcTask Outputs/MAIN.enable_cmd[107] <-> Control process data mapping/enable
//     PlcTask Outputs/MAIN.force_cmd_X[107] <-> Control process data mapping/force_sp_X
//     PlcTask Outputs/MAIN.force_cmd_Y[107] <-> Control process data mapping/force_sp_Y
//     PlcTask Outputs/MAIN.force_cmd_Z[107] <-> Control process data mapping/force_sp_Z
//     PlcTask Outputs/MAIN.msthb[115] <-> Control process data mapping/msthb
//   SAsetGains/SAsetGains Instance <-> Device 1 (EtherCAT)/Box 114 (m1eph)/Box 116 (m1sa)
//     PlcTask Inputs/MAIN.cloop_stat[108] <-> Status process data mapping/close_loop
//     PlcTask Inputs/MAIN.enable_stat[108] <-> Status process data mapping/enable
//     PlcTask Inputs/MAIN.force_rb_X[108] <-> Status process data mapping/force_rb_X
//     PlcTask Inputs/MAIN.force_rb_Y[108] <-> Status process data mapping/force_rb_Y
//     PlcTask Inputs/MAIN.force_rb_Z[108] <-> Status process data mapping/force_rb_Z
//     PlcTask Inputs/MAIN.force_sp_X[108] <-> Status process data mapping/force_sp_X
//     PlcTask Inputs/MAIN.force_sp_Y[108] <-> Status process data mapping/force_sp_Y
//     PlcTask Inputs/MAIN.force_sp_Z[108] <-> Status process data mapping/force_sp_Z
//     PlcTask Inputs/MAIN.pwm1[108] <-> Status process data mapping/pwm1
//     PlcTask Inputs/MAIN.pwm2[108] <-> Status process data mapping/pwm2
//     PlcTask Inputs/MAIN.pwm3[108] <-> Status process data mapping/pwm3
//     PlcTask Outputs/MAIN.enable_cmd[108] <-> Control process data mapping/enable
//     PlcTask Outputs/MAIN.force_cmd_X[108] <-> Control process data mapping/force_sp_X
//     PlcTask Outputs/MAIN.force_cmd_Y[108] <-> Control process data mapping/force_sp_Y
//     PlcTask Outputs/MAIN.force_cmd_Z[108] <-> Control process data mapping/force_sp_Z
//     PlcTask Outputs/MAIN.msthb[116] <-> Control process data mapping/msthb
//   SAsetGains/SAsetGains Instance <-> Device 1 (EtherCAT)/Box 114 (m1eph)/Box 117 (m1sa)
//     PlcTask Inputs/MAIN.cloop_stat[109] <-> Status process data mapping/close_loop
//     PlcTask Inputs/MAIN.enable_stat[109] <-> Status process data mapping/enable
//     PlcTask Inputs/MAIN.force_rb_X[109] <-> Status process data mapping/force_rb_X
//     PlcTask Inputs/MAIN.force_rb_Y[109] <-> Status process data mapping/force_rb_Y
//     PlcTask Inputs/MAIN.force_rb_Z[109] <-> Status process data mapping/force_rb_Z
//     PlcTask Inputs/MAIN.force_sp_X[109] <-> Status process data mapping/force_sp_X
//     PlcTask Inputs/MAIN.force_sp_Y[109] <-> Status process data mapping/force_sp_Y
//     PlcTask Inputs/MAIN.force_sp_Z[109] <-> Status process data mapping/force_sp_Z
//     PlcTask Inputs/MAIN.pwm1[109] <-> Status process data mapping/pwm1
//     PlcTask Inputs/MAIN.pwm2[109] <-> Status process data mapping/pwm2
//     PlcTask Inputs/MAIN.pwm3[109] <-> Status process data mapping/pwm3
//     PlcTask Outputs/MAIN.enable_cmd[109] <-> Control process data mapping/enable
//     PlcTask Outputs/MAIN.force_cmd_X[109] <-> Control process data mapping/force_sp_X
//     PlcTask Outputs/MAIN.force_cmd_Y[109] <-> Control process data mapping/force_sp_Y
//     PlcTask Outputs/MAIN.force_cmd_Z[109] <-> Control process data mapping/force_sp_Z
//     PlcTask Outputs/MAIN.msthb[117] <-> Control process data mapping/msthb
//   SAsetGains/SAsetGains Instance <-> Device 1 (EtherCAT)/Box 114 (m1eph)/Box 118 (m1sa)
//     PlcTask Inputs/MAIN.cloop_stat[110] <-> Status process data mapping/close_loop
//     PlcTask Inputs/MAIN.enable_stat[110] <-> Status process data mapping/enable
//     PlcTask Inputs/MAIN.force_rb_X[110] <-> Status process data mapping/force_rb_X
//     PlcTask Inputs/MAIN.force_rb_Y[110] <-> Status process data mapping/force_rb_Y
//     PlcTask Inputs/MAIN.force_rb_Z[110] <-> Status process data mapping/force_rb_Z
//     PlcTask Inputs/MAIN.force_sp_X[110] <-> Status process data mapping/force_sp_X
//     PlcTask Inputs/MAIN.force_sp_Y[110] <-> Status process data mapping/force_sp_Y
//     PlcTask Inputs/MAIN.force_sp_Z[110] <-> Status process data mapping/force_sp_Z
//     PlcTask Inputs/MAIN.pwm1[110] <-> Status process data mapping/pwm1
//     PlcTask Inputs/MAIN.pwm2[110] <-> Status process data mapping/pwm2
//     PlcTask Inputs/MAIN.pwm3[110] <-> Status process data mapping/pwm3
//     PlcTask Outputs/MAIN.enable_cmd[110] <-> Control process data mapping/enable
//     PlcTask Outputs/MAIN.force_cmd_X[110] <-> Control process data mapping/force_sp_X
//     PlcTask Outputs/MAIN.force_cmd_Y[110] <-> Control process data mapping/force_sp_Y
//     PlcTask Outputs/MAIN.force_cmd_Z[110] <-> Control process data mapping/force_sp_Z
//     PlcTask Outputs/MAIN.msthb[118] <-> Control process data mapping/msthb
//   SAsetGains/SAsetGains Instance <-> Device 1 (EtherCAT)/Box 114 (m1eph)/Box 119 (m1sa)
//     PlcTask Inputs/MAIN.cloop_stat[111] <-> Status process data mapping/close_loop
//     PlcTask Inputs/MAIN.enable_stat[111] <-> Status process data mapping/enable
//     PlcTask Inputs/MAIN.force_rb_X[111] <-> Status process data mapping/force_rb_X
//     PlcTask Inputs/MAIN.force_rb_Y[111] <-> Status process data mapping/force_rb_Y
//     PlcTask Inputs/MAIN.force_rb_Z[111] <-> Status process data mapping/force_rb_Z
//     PlcTask Inputs/MAIN.force_sp_X[111] <-> Status process data mapping/force_sp_X
//     PlcTask Inputs/MAIN.force_sp_Y[111] <-> Status process data mapping/force_sp_Y
//     PlcTask Inputs/MAIN.force_sp_Z[111] <-> Status process data mapping/force_sp_Z
//     PlcTask Inputs/MAIN.pwm1[111] <-> Status process data mapping/pwm1
//     PlcTask Inputs/MAIN.pwm2[111] <-> Status process data mapping/pwm2
//     PlcTask Inputs/MAIN.pwm3[111] <-> Status process data mapping/pwm3
//     PlcTask Outputs/MAIN.enable_cmd[111] <-> Control process data mapping/enable
//     PlcTask Outputs/MAIN.force_cmd_X[111] <-> Control process data mapping/force_sp_X
//     PlcTask Outputs/MAIN.force_cmd_Y[111] <-> Control process data mapping/force_sp_Y
//     PlcTask Outputs/MAIN.force_cmd_Z[111] <-> Control process data mapping/force_sp_Z
//     PlcTask Outputs/MAIN.msthb[119] <-> Control process data mapping/msthb
//   SAsetGains/SAsetGains Instance <-> Device 1 (EtherCAT)/Box 114 (m1eph)/Box 120 (m1sa)
//     PlcTask Inputs/MAIN.cloop_stat[112] <-> Status process data mapping/close_loop
//     PlcTask Inputs/MAIN.enable_stat[112] <-> Status process data mapping/enable
//     PlcTask Inputs/MAIN.force_rb_X[112] <-> Status process data mapping/force_rb_X
//     PlcTask Inputs/MAIN.force_rb_Y[112] <-> Status process data mapping/force_rb_Y
//     PlcTask Inputs/MAIN.force_rb_Z[112] <-> Status process data mapping/force_rb_Z
//     PlcTask Inputs/MAIN.force_sp_X[112] <-> Status process data mapping/force_sp_X
//     PlcTask Inputs/MAIN.force_sp_Y[112] <-> Status process data mapping/force_sp_Y
//     PlcTask Inputs/MAIN.force_sp_Z[112] <-> Status process data mapping/force_sp_Z
//     PlcTask Inputs/MAIN.pwm1[112] <-> Status process data mapping/pwm1
//     PlcTask Inputs/MAIN.pwm2[112] <-> Status process data mapping/pwm2
//     PlcTask Inputs/MAIN.pwm3[112] <-> Status process data mapping/pwm3
//     PlcTask Outputs/MAIN.enable_cmd[112] <-> Control process data mapping/enable
//     PlcTask Outputs/MAIN.force_cmd_X[112] <-> Control process data mapping/force_sp_X
//     PlcTask Outputs/MAIN.force_cmd_Y[112] <-> Control process data mapping/force_sp_Y
//     PlcTask Outputs/MAIN.force_cmd_Z[112] <-> Control process data mapping/force_sp_Z
//     PlcTask Outputs/MAIN.msthb[120] <-> Control process data mapping/msthb
//   SAsetGains/SAsetGains Instance <-> Device 1 (EtherCAT)/Box 114 (m1eph)/Box 121 (m1sa)
//     PlcTask Inputs/MAIN.cloop_stat[113] <-> Status process data mapping/close_loop
//     PlcTask Inputs/MAIN.enable_stat[113] <-> Status process data mapping/enable
//     PlcTask Inputs/MAIN.force_rb_X[113] <-> Status process data mapping/force_rb_X
//     PlcTask Inputs/MAIN.force_rb_Y[113] <-> Status process data mapping/force_rb_Y
//     PlcTask Inputs/MAIN.force_rb_Z[113] <-> Status process data mapping/force_rb_Z
//     PlcTask Inputs/MAIN.force_sp_X[113] <-> Status process data mapping/force_sp_X
//     PlcTask Inputs/MAIN.force_sp_Y[113] <-> Status process data mapping/force_sp_Y
//     PlcTask Inputs/MAIN.force_sp_Z[113] <-> Status process data mapping/force_sp_Z
//     PlcTask Inputs/MAIN.pwm1[113] <-> Status process data mapping/pwm1
//     PlcTask Inputs/MAIN.pwm2[113] <-> Status process data mapping/pwm2
//     PlcTask Inputs/MAIN.pwm3[113] <-> Status process data mapping/pwm3
//     PlcTask Outputs/MAIN.enable_cmd[113] <-> Control process data mapping/enable
//     PlcTask Outputs/MAIN.force_cmd_X[113] <-> Control process data mapping/force_sp_X
//     PlcTask Outputs/MAIN.force_cmd_Y[113] <-> Control process data mapping/force_sp_Y
//     PlcTask Outputs/MAIN.force_cmd_Z[113] <-> Control process data mapping/force_sp_Z
//     PlcTask Outputs/MAIN.msthb[121] <-> Control process data mapping/msthb
//   SAsetGains/SAsetGains Instance <-> Device 1 (EtherCAT)/Box 114 (m1eph)/Box 122 (m1sa)
//     PlcTask Inputs/MAIN.cloop_stat[114] <-> Status process data mapping/close_loop
//     PlcTask Inputs/MAIN.enable_stat[114] <-> Status process data mapping/enable
//     PlcTask Inputs/MAIN.force_rb_X[114] <-> Status process data mapping/force_rb_X
//     PlcTask Inputs/MAIN.force_rb_Y[114] <-> Status process data mapping/force_rb_Y
//     PlcTask Inputs/MAIN.force_rb_Z[114] <-> Status process data mapping/force_rb_Z
//     PlcTask Inputs/MAIN.force_sp_X[114] <-> Status process data mapping/force_sp_X
//     PlcTask Inputs/MAIN.force_sp_Y[114] <-> Status process data mapping/force_sp_Y
//     PlcTask Inputs/MAIN.force_sp_Z[114] <-> Status process data mapping/force_sp_Z
//     PlcTask Inputs/MAIN.pwm1[114] <-> Status process data mapping/pwm1
//     PlcTask Inputs/MAIN.pwm2[114] <-> Status process data mapping/pwm2
//     PlcTask Inputs/MAIN.pwm3[114] <-> Status process data mapping/pwm3
//     PlcTask Outputs/MAIN.enable_cmd[114] <-> Control process data mapping/enable
//     PlcTask Outputs/MAIN.force_cmd_X[114] <-> Control process data mapping/force_sp_X
//     PlcTask Outputs/MAIN.force_cmd_Y[114] <-> Control process data mapping/force_sp_Y
//     PlcTask Outputs/MAIN.force_cmd_Z[114] <-> Control process data mapping/force_sp_Z
//     PlcTask Outputs/MAIN.msthb[122] <-> Control process data mapping/msthb
//   SAsetGains/SAsetGains Instance <-> Device 1 (EtherCAT)/Box 114 (m1eph)/Box 123 (m1sa)
//     PlcTask Inputs/MAIN.cloop_stat[115] <-> Status process data mapping/close_loop
//     PlcTask Inputs/MAIN.enable_stat[115] <-> Status process data mapping/enable
//     PlcTask Inputs/MAIN.force_rb_X[115] <-> Status process data mapping/force_rb_X
//     PlcTask Inputs/MAIN.force_rb_Y[115] <-> Status process data mapping/force_rb_Y
//     PlcTask Inputs/MAIN.force_rb_Z[115] <-> Status process data mapping/force_rb_Z
//     PlcTask Inputs/MAIN.force_sp_X[115] <-> Status process data mapping/force_sp_X
//     PlcTask Inputs/MAIN.force_sp_Y[115] <-> Status process data mapping/force_sp_Y
//     PlcTask Inputs/MAIN.force_sp_Z[115] <-> Status process data mapping/force_sp_Z
//     PlcTask Inputs/MAIN.pwm1[115] <-> Status process data mapping/pwm1
//     PlcTask Inputs/MAIN.pwm2[115] <-> Status process data mapping/pwm2
//     PlcTask Inputs/MAIN.pwm3[115] <-> Status process data mapping/pwm3
//     PlcTask Outputs/MAIN.enable_cmd[115] <-> Control process data mapping/enable
//     PlcTask Outputs/MAIN.force_cmd_X[115] <-> Control process data mapping/force_sp_X
//     PlcTask Outputs/MAIN.force_cmd_Y[115] <-> Control process data mapping/force_sp_Y
//     PlcTask Outputs/MAIN.force_cmd_Z[115] <-> Control process data mapping/force_sp_Z
//     PlcTask Outputs/MAIN.msthb[123] <-> Control process data mapping/msthb
//   SAsetGains/SAsetGains Instance <-> Device 1 (EtherCAT)/Box 114 (m1eph)/Box 124 (m1sa)
//     PlcTask Inputs/MAIN.cloop_stat[116] <-> Status process data mapping/close_loop
//     PlcTask Inputs/MAIN.enable_stat[116] <-> Status process data mapping/enable
//     PlcTask Inputs/MAIN.force_rb_X[116] <-> Status process data mapping/force_rb_X
//     PlcTask Inputs/MAIN.force_rb_Y[116] <-> Status process data mapping/force_rb_Y
//     PlcTask Inputs/MAIN.force_rb_Z[116] <-> Status process data mapping/force_rb_Z
//     PlcTask Inputs/MAIN.force_sp_X[116] <-> Status process data mapping/force_sp_X
//     PlcTask Inputs/MAIN.force_sp_Y[116] <-> Status process data mapping/force_sp_Y
//     PlcTask Inputs/MAIN.force_sp_Z[116] <-> Status process data mapping/force_sp_Z
//     PlcTask Inputs/MAIN.pwm1[116] <-> Status process data mapping/pwm1
//     PlcTask Inputs/MAIN.pwm2[116] <-> Status process data mapping/pwm2
//     PlcTask Inputs/MAIN.pwm3[116] <-> Status process data mapping/pwm3
//     PlcTask Outputs/MAIN.enable_cmd[116] <-> Control process data mapping/enable
//     PlcTask Outputs/MAIN.force_cmd_X[116] <-> Control process data mapping/force_sp_X
//     PlcTask Outputs/MAIN.force_cmd_Y[116] <-> Control process data mapping/force_sp_Y
//     PlcTask Outputs/MAIN.force_cmd_Z[116] <-> Control process data mapping/force_sp_Z
//     PlcTask Outputs/MAIN.msthb[124] <-> Control process data mapping/msthb
//   SAsetGains/SAsetGains Instance <-> Device 1 (EtherCAT)/Box 114 (m1eph)/Box 125 (m1sa)
//     PlcTask Inputs/MAIN.cloop_stat[117] <-> Status process data mapping/close_loop
//     PlcTask Inputs/MAIN.enable_stat[117] <-> Status process data mapping/enable
//     PlcTask Inputs/MAIN.force_rb_X[117] <-> Status process data mapping/force_rb_X
//     PlcTask Inputs/MAIN.force_rb_Y[117] <-> Status process data mapping/force_rb_Y
//     PlcTask Inputs/MAIN.force_rb_Z[117] <-> Status process data mapping/force_rb_Z
//     PlcTask Inputs/MAIN.force_sp_X[117] <-> Status process data mapping/force_sp_X
//     PlcTask Inputs/MAIN.force_sp_Y[117] <-> Status process data mapping/force_sp_Y
//     PlcTask Inputs/MAIN.force_sp_Z[117] <-> Status process data mapping/force_sp_Z
//     PlcTask Inputs/MAIN.pwm1[117] <-> Status process data mapping/pwm1
//     PlcTask Inputs/MAIN.pwm2[117] <-> Status process data mapping/pwm2
//     PlcTask Inputs/MAIN.pwm3[117] <-> Status process data mapping/pwm3
//     PlcTask Outputs/MAIN.enable_cmd[117] <-> Control process data mapping/enable
//     PlcTask Outputs/MAIN.force_cmd_X[117] <-> Control process data mapping/force_sp_X
//     PlcTask Outputs/MAIN.force_cmd_Y[117] <-> Control process data mapping/force_sp_Y
//     PlcTask Outputs/MAIN.force_cmd_Z[117] <-> Control process data mapping/force_sp_Z
//     PlcTask Outputs/MAIN.msthb[125] <-> Control process data mapping/msthb
//   SAsetGains/SAsetGains Instance <-> Device 1 (EtherCAT)/Box 114 (m1eph)/Box 126 (m1sa)
//     PlcTask Inputs/MAIN.cloop_stat[118] <-> Status process data mapping/close_loop
//     PlcTask Inputs/MAIN.enable_stat[118] <-> Status process data mapping/enable
//     PlcTask Inputs/MAIN.force_rb_X[118] <-> Status process data mapping/force_rb_X
//     PlcTask Inputs/MAIN.force_rb_Y[118] <-> Status process data mapping/force_rb_Y
//     PlcTask Inputs/MAIN.force_rb_Z[118] <-> Status process data mapping/force_rb_Z
//     PlcTask Inputs/MAIN.force_sp_X[118] <-> Status process data mapping/force_sp_X
//     PlcTask Inputs/MAIN.force_sp_Y[118] <-> Status process data mapping/force_sp_Y
//     PlcTask Inputs/MAIN.force_sp_Z[118] <-> Status process data mapping/force_sp_Z
//     PlcTask Inputs/MAIN.pwm1[118] <-> Status process data mapping/pwm1
//     PlcTask Inputs/MAIN.pwm2[118] <-> Status process data mapping/pwm2
//     PlcTask Inputs/MAIN.pwm3[118] <-> Status process data mapping/pwm3
//     PlcTask Outputs/MAIN.enable_cmd[118] <-> Control process data mapping/enable
//     PlcTask Outputs/MAIN.force_cmd_X[118] <-> Control process data mapping/force_sp_X
//     PlcTask Outputs/MAIN.force_cmd_Y[118] <-> Control process data mapping/force_sp_Y
//     PlcTask Outputs/MAIN.force_cmd_Z[118] <-> Control process data mapping/force_sp_Z
//     PlcTask Outputs/MAIN.msthb[126] <-> Control process data mapping/msthb
//   SAsetGains/SAsetGains Instance <-> Device 1 (EtherCAT)/Box 114 (m1eph)/Box 127 (m1sa)
//     PlcTask Inputs/MAIN.cloop_stat[119] <-> Status process data mapping/close_loop
//     PlcTask Inputs/MAIN.enable_stat[119] <-> Status process data mapping/enable
//     PlcTask Inputs/MAIN.force_rb_X[119] <-> Status process data mapping/force_rb_X
//     PlcTask Inputs/MAIN.force_rb_Y[119] <-> Status process data mapping/force_rb_Y
//     PlcTask Inputs/MAIN.force_rb_Z[119] <-> Status process data mapping/force_rb_Z
//     PlcTask Inputs/MAIN.force_sp_X[119] <-> Status process data mapping/force_sp_X
//     PlcTask Inputs/MAIN.force_sp_Y[119] <-> Status process data mapping/force_sp_Y
//     PlcTask Inputs/MAIN.force_sp_Z[119] <-> Status process data mapping/force_sp_Z
//     PlcTask Inputs/MAIN.pwm1[119] <-> Status process data mapping/pwm1
//     PlcTask Inputs/MAIN.pwm2[119] <-> Status process data mapping/pwm2
//     PlcTask Inputs/MAIN.pwm3[119] <-> Status process data mapping/pwm3
//     PlcTask Outputs/MAIN.enable_cmd[119] <-> Control process data mapping/enable
//     PlcTask Outputs/MAIN.force_cmd_X[119] <-> Control process data mapping/force_sp_X
//     PlcTask Outputs/MAIN.force_cmd_Y[119] <-> Control process data mapping/force_sp_Y
//     PlcTask Outputs/MAIN.force_cmd_Z[119] <-> Control process data mapping/force_sp_Z
//     PlcTask Outputs/MAIN.msthb[127] <-> Control process data mapping/msthb
//   SAsetGains/SAsetGains Instance <-> Device 1 (EtherCAT)/Box 114 (m1eph)/Box 128 (m1sa)
//     PlcTask Inputs/MAIN.cloop_stat[120] <-> Status process data mapping/close_loop
//     PlcTask Inputs/MAIN.enable_stat[120] <-> Status process data mapping/enable
//     PlcTask Inputs/MAIN.force_rb_X[120] <-> Status process data mapping/force_rb_X
//     PlcTask Inputs/MAIN.force_rb_Y[120] <-> Status process data mapping/force_rb_Y
//     PlcTask Inputs/MAIN.force_rb_Z[120] <-> Status process data mapping/force_rb_Z
//     PlcTask Inputs/MAIN.force_sp_X[120] <-> Status process data mapping/force_sp_X
//     PlcTask Inputs/MAIN.force_sp_Y[120] <-> Status process data mapping/force_sp_Y
//     PlcTask Inputs/MAIN.force_sp_Z[120] <-> Status process data mapping/force_sp_Z
//     PlcTask Inputs/MAIN.pwm1[120] <-> Status process data mapping/pwm1
//     PlcTask Inputs/MAIN.pwm2[120] <-> Status process data mapping/pwm2
//     PlcTask Inputs/MAIN.pwm3[120] <-> Status process data mapping/pwm3
//     PlcTask Outputs/MAIN.enable_cmd[120] <-> Control process data mapping/enable
//     PlcTask Outputs/MAIN.force_cmd_X[120] <-> Control process data mapping/force_sp_X
//     PlcTask Outputs/MAIN.force_cmd_Y[120] <-> Control process data mapping/force_sp_Y
//     PlcTask Outputs/MAIN.force_cmd_Z[120] <-> Control process data mapping/force_sp_Z
//     PlcTask Outputs/MAIN.msthb[128] <-> Control process data mapping/msthb
//   SAsetGains/SAsetGains Instance <-> Device 1 (EtherCAT)/Box 114 (m1eph)/Box 129 (m1sa)
//     PlcTask Inputs/MAIN.cloop_stat[121] <-> Status process data mapping/close_loop
//     PlcTask Inputs/MAIN.enable_stat[121] <-> Status process data mapping/enable
//     PlcTask Inputs/MAIN.force_rb_X[121] <-> Status process data mapping/force_rb_X
//     PlcTask Inputs/MAIN.force_rb_Y[121] <-> Status process data mapping/force_rb_Y
//     PlcTask Inputs/MAIN.force_rb_Z[121] <-> Status process data mapping/force_rb_Z
//     PlcTask Inputs/MAIN.force_sp_X[121] <-> Status process data mapping/force_sp_X
//     PlcTask Inputs/MAIN.force_sp_Y[121] <-> Status process data mapping/force_sp_Y
//     PlcTask Inputs/MAIN.force_sp_Z[121] <-> Status process data mapping/force_sp_Z
//     PlcTask Inputs/MAIN.pwm1[121] <-> Status process data mapping/pwm1
//     PlcTask Inputs/MAIN.pwm2[121] <-> Status process data mapping/pwm2
//     PlcTask Inputs/MAIN.pwm3[121] <-> Status process data mapping/pwm3
//     PlcTask Outputs/MAIN.enable_cmd[121] <-> Control process data mapping/enable
//     PlcTask Outputs/MAIN.force_cmd_X[121] <-> Control process data mapping/force_sp_X
//     PlcTask Outputs/MAIN.force_cmd_Y[121] <-> Control process data mapping/force_sp_Y
//     PlcTask Outputs/MAIN.force_cmd_Z[121] <-> Control process data mapping/force_sp_Z
//     PlcTask Outputs/MAIN.msthb[129] <-> Control process data mapping/msthb
//   SAsetGains/SAsetGains Instance <-> Device 1 (EtherCAT)/Box 114 (m1eph)/Box 130 (m1sa)
//     PlcTask Inputs/MAIN.cloop_stat[122] <-> Status process data mapping/close_loop
//     PlcTask Inputs/MAIN.enable_stat[122] <-> Status process data mapping/enable
//     PlcTask Inputs/MAIN.force_rb_X[122] <-> Status process data mapping/force_rb_X
//     PlcTask Inputs/MAIN.force_rb_Y[122] <-> Status process data mapping/force_rb_Y
//     PlcTask Inputs/MAIN.force_rb_Z[122] <-> Status process data mapping/force_rb_Z
//     PlcTask Inputs/MAIN.force_sp_X[122] <-> Status process data mapping/force_sp_X
//     PlcTask Inputs/MAIN.force_sp_Y[122] <-> Status process data mapping/force_sp_Y
//     PlcTask Inputs/MAIN.force_sp_Z[122] <-> Status process data mapping/force_sp_Z
//     PlcTask Inputs/MAIN.pwm1[122] <-> Status process data mapping/pwm1
//     PlcTask Inputs/MAIN.pwm2[122] <-> Status process data mapping/pwm2
//     PlcTask Inputs/MAIN.pwm3[122] <-> Status process data mapping/pwm3
//     PlcTask Outputs/MAIN.enable_cmd[122] <-> Control process data mapping/enable
//     PlcTask Outputs/MAIN.force_cmd_X[122] <-> Control process data mapping/force_sp_X
//     PlcTask Outputs/MAIN.force_cmd_Y[122] <-> Control process data mapping/force_sp_Y
//     PlcTask Outputs/MAIN.force_cmd_Z[122] <-> Control process data mapping/force_sp_Z
//     PlcTask Outputs/MAIN.msthb[130] <-> Control process data mapping/msthb
//   SAsetGains/SAsetGains Instance <-> Device 1 (EtherCAT)/Box 131 (m1eph)
//     PlcTask Outputs/MAIN.msthb[131] <-> Control process data mapping/msthb
//   SAsetGains/SAsetGains Instance <-> Device 1 (EtherCAT)/Box 131 (m1eph)/Box 132 (m1sa)
//     PlcTask Inputs/MAIN.cloop_stat[123] <-> Status process data mapping/close_loop
//     PlcTask Inputs/MAIN.enable_stat[123] <-> Status process data mapping/enable
//     PlcTask Inputs/MAIN.force_rb_X[123] <-> Status process data mapping/force_rb_X
//     PlcTask Inputs/MAIN.force_rb_Y[123] <-> Status process data mapping/force_rb_Y
//     PlcTask Inputs/MAIN.force_rb_Z[123] <-> Status process data mapping/force_rb_Z
//     PlcTask Inputs/MAIN.force_sp_X[123] <-> Status process data mapping/force_sp_X
//     PlcTask Inputs/MAIN.force_sp_Y[123] <-> Status process data mapping/force_sp_Y
//     PlcTask Inputs/MAIN.force_sp_Z[123] <-> Status process data mapping/force_sp_Z
//     PlcTask Inputs/MAIN.pwm1[123] <-> Status process data mapping/pwm1
//     PlcTask Inputs/MAIN.pwm2[123] <-> Status process data mapping/pwm2
//     PlcTask Inputs/MAIN.pwm3[123] <-> Status process data mapping/pwm3
//     PlcTask Outputs/MAIN.enable_cmd[123] <-> Control process data mapping/enable
//     PlcTask Outputs/MAIN.force_cmd_X[123] <-> Control process data mapping/force_sp_X
//     PlcTask Outputs/MAIN.force_cmd_Y[123] <-> Control process data mapping/force_sp_Y
//     PlcTask Outputs/MAIN.force_cmd_Z[123] <-> Control process data mapping/force_sp_Z
//     PlcTask Outputs/MAIN.msthb[132] <-> Control process data mapping/msthb
//   SAsetGains/SAsetGains Instance <-> Device 1 (EtherCAT)/Box 131 (m1eph)/Box 133 (m1sa)
//     PlcTask Inputs/MAIN.cloop_stat[124] <-> Status process data mapping/close_loop
//     PlcTask Inputs/MAIN.enable_stat[124] <-> Status process data mapping/enable
//     PlcTask Inputs/MAIN.force_rb_X[124] <-> Status process data mapping/force_rb_X
//     PlcTask Inputs/MAIN.force_rb_Y[124] <-> Status process data mapping/force_rb_Y
//     PlcTask Inputs/MAIN.force_rb_Z[124] <-> Status process data mapping/force_rb_Z
//     PlcTask Inputs/MAIN.force_sp_X[124] <-> Status process data mapping/force_sp_X
//     PlcTask Inputs/MAIN.force_sp_Y[124] <-> Status process data mapping/force_sp_Y
//     PlcTask Inputs/MAIN.force_sp_Z[124] <-> Status process data mapping/force_sp_Z
//     PlcTask Inputs/MAIN.pwm1[124] <-> Status process data mapping/pwm1
//     PlcTask Inputs/MAIN.pwm2[124] <-> Status process data mapping/pwm2
//     PlcTask Inputs/MAIN.pwm3[124] <-> Status process data mapping/pwm3
//     PlcTask Outputs/MAIN.enable_cmd[124] <-> Control process data mapping/enable
//     PlcTask Outputs/MAIN.force_cmd_X[124] <-> Control process data mapping/force_sp_X
//     PlcTask Outputs/MAIN.force_cmd_Y[124] <-> Control process data mapping/force_sp_Y
//     PlcTask Outputs/MAIN.force_cmd_Z[124] <-> Control process data mapping/force_sp_Z
//     PlcTask Outputs/MAIN.msthb[133] <-> Control process data mapping/msthb
//   SAsetGains/SAsetGains Instance <-> Device 1 (EtherCAT)/Box 131 (m1eph)/Box 134 (m1sa)
//     PlcTask Inputs/MAIN.cloop_stat[125] <-> Status process data mapping/close_loop
//     PlcTask Inputs/MAIN.enable_stat[125] <-> Status process data mapping/enable
//     PlcTask Inputs/MAIN.force_rb_X[125] <-> Status process data mapping/force_rb_X
//     PlcTask Inputs/MAIN.force_rb_Y[125] <-> Status process data mapping/force_rb_Y
//     PlcTask Inputs/MAIN.force_rb_Z[125] <-> Status process data mapping/force_rb_Z
//     PlcTask Inputs/MAIN.force_sp_X[125] <-> Status process data mapping/force_sp_X
//     PlcTask Inputs/MAIN.force_sp_Y[125] <-> Status process data mapping/force_sp_Y
//     PlcTask Inputs/MAIN.force_sp_Z[125] <-> Status process data mapping/force_sp_Z
//     PlcTask Inputs/MAIN.pwm1[125] <-> Status process data mapping/pwm1
//     PlcTask Inputs/MAIN.pwm2[125] <-> Status process data mapping/pwm2
//     PlcTask Inputs/MAIN.pwm3[125] <-> Status process data mapping/pwm3
//     PlcTask Outputs/MAIN.enable_cmd[125] <-> Control process data mapping/enable
//     PlcTask Outputs/MAIN.force_cmd_X[125] <-> Control process data mapping/force_sp_X
//     PlcTask Outputs/MAIN.force_cmd_Y[125] <-> Control process data mapping/force_sp_Y
//     PlcTask Outputs/MAIN.force_cmd_Z[125] <-> Control process data mapping/force_sp_Z
//     PlcTask Outputs/MAIN.msthb[134] <-> Control process data mapping/msthb
//   SAsetGains/SAsetGains Instance <-> Device 1 (EtherCAT)/Box 131 (m1eph)/Box 135 (m1sa)
//     PlcTask Inputs/MAIN.cloop_stat[126] <-> Status process data mapping/close_loop
//     PlcTask Inputs/MAIN.enable_stat[126] <-> Status process data mapping/enable
//     PlcTask Inputs/MAIN.force_rb_X[126] <-> Status process data mapping/force_rb_X
//     PlcTask Inputs/MAIN.force_rb_Y[126] <-> Status process data mapping/force_rb_Y
//     PlcTask Inputs/MAIN.force_rb_Z[126] <-> Status process data mapping/force_rb_Z
//     PlcTask Inputs/MAIN.force_sp_X[126] <-> Status process data mapping/force_sp_X
//     PlcTask Inputs/MAIN.force_sp_Y[126] <-> Status process data mapping/force_sp_Y
//     PlcTask Inputs/MAIN.force_sp_Z[126] <-> Status process data mapping/force_sp_Z
//     PlcTask Inputs/MAIN.pwm1[126] <-> Status process data mapping/pwm1
//     PlcTask Inputs/MAIN.pwm2[126] <-> Status process data mapping/pwm2
//     PlcTask Inputs/MAIN.pwm3[126] <-> Status process data mapping/pwm3
//     PlcTask Outputs/MAIN.enable_cmd[126] <-> Control process data mapping/enable
//     PlcTask Outputs/MAIN.force_cmd_X[126] <-> Control process data mapping/force_sp_X
//     PlcTask Outputs/MAIN.force_cmd_Y[126] <-> Control process data mapping/force_sp_Y
//     PlcTask Outputs/MAIN.force_cmd_Z[126] <-> Control process data mapping/force_sp_Z
//     PlcTask Outputs/MAIN.msthb[135] <-> Control process data mapping/msthb
//   SAsetGains/SAsetGains Instance <-> Device 1 (EtherCAT)/Box 131 (m1eph)/Box 136 (m1sa)
//     PlcTask Inputs/MAIN.cloop_stat[127] <-> Status process data mapping/close_loop
//     PlcTask Inputs/MAIN.enable_stat[127] <-> Status process data mapping/enable
//     PlcTask Inputs/MAIN.force_rb_X[127] <-> Status process data mapping/force_rb_X
//     PlcTask Inputs/MAIN.force_rb_Y[127] <-> Status process data mapping/force_rb_Y
//     PlcTask Inputs/MAIN.force_rb_Z[127] <-> Status process data mapping/force_rb_Z
//     PlcTask Inputs/MAIN.force_sp_X[127] <-> Status process data mapping/force_sp_X
//     PlcTask Inputs/MAIN.force_sp_Y[127] <-> Status process data mapping/force_sp_Y
//     PlcTask Inputs/MAIN.force_sp_Z[127] <-> Status process data mapping/force_sp_Z
//     PlcTask Inputs/MAIN.pwm1[127] <-> Status process data mapping/pwm1
//     PlcTask Inputs/MAIN.pwm2[127] <-> Status process data mapping/pwm2
//     PlcTask Inputs/MAIN.pwm3[127] <-> Status process data mapping/pwm3
//     PlcTask Outputs/MAIN.enable_cmd[127] <-> Control process data mapping/enable
//     PlcTask Outputs/MAIN.force_cmd_X[127] <-> Control process data mapping/force_sp_X
//     PlcTask Outputs/MAIN.force_cmd_Y[127] <-> Control process data mapping/force_sp_Y
//     PlcTask Outputs/MAIN.force_cmd_Z[127] <-> Control process data mapping/force_sp_Z
//     PlcTask Outputs/MAIN.msthb[136] <-> Control process data mapping/msthb
//   SAsetGains/SAsetGains Instance <-> Device 1 (EtherCAT)/Box 131 (m1eph)/Box 137 (m1sa)
//     PlcTask Inputs/MAIN.cloop_stat[128] <-> Status process data mapping/close_loop
//     PlcTask Inputs/MAIN.enable_stat[128] <-> Status process data mapping/enable
//     PlcTask Inputs/MAIN.force_rb_X[128] <-> Status process data mapping/force_rb_X
//     PlcTask Inputs/MAIN.force_rb_Y[128] <-> Status process data mapping/force_rb_Y
//     PlcTask Inputs/MAIN.force_rb_Z[128] <-> Status process data mapping/force_rb_Z
//     PlcTask Inputs/MAIN.force_sp_X[128] <-> Status process data mapping/force_sp_X
//     PlcTask Inputs/MAIN.force_sp_Y[128] <-> Status process data mapping/force_sp_Y
//     PlcTask Inputs/MAIN.force_sp_Z[128] <-> Status process data mapping/force_sp_Z
//     PlcTask Inputs/MAIN.pwm1[128] <-> Status process data mapping/pwm1
//     PlcTask Inputs/MAIN.pwm2[128] <-> Status process data mapping/pwm2
//     PlcTask Inputs/MAIN.pwm3[128] <-> Status process data mapping/pwm3
//     PlcTask Outputs/MAIN.enable_cmd[128] <-> Control process data mapping/enable
//     PlcTask Outputs/MAIN.force_cmd_X[128] <-> Control process data mapping/force_sp_X
//     PlcTask Outputs/MAIN.force_cmd_Y[128] <-> Control process data mapping/force_sp_Y
//     PlcTask Outputs/MAIN.force_cmd_Z[128] <-> Control process data mapping/force_sp_Z
//     PlcTask Outputs/MAIN.msthb[137] <-> Control process data mapping/msthb
//   SAsetGains/SAsetGains Instance <-> Device 1 (EtherCAT)/Box 131 (m1eph)/Box 138 (m1sa)
//     PlcTask Inputs/MAIN.cloop_stat[129] <-> Status process data mapping/close_loop
//     PlcTask Inputs/MAIN.enable_stat[129] <-> Status process data mapping/enable
//     PlcTask Inputs/MAIN.force_rb_X[129] <-> Status process data mapping/force_rb_X
//     PlcTask Inputs/MAIN.force_rb_Y[129] <-> Status process data mapping/force_rb_Y
//     PlcTask Inputs/MAIN.force_rb_Z[129] <-> Status process data mapping/force_rb_Z
//     PlcTask Inputs/MAIN.force_sp_X[129] <-> Status process data mapping/force_sp_X
//     PlcTask Inputs/MAIN.force_sp_Y[129] <-> Status process data mapping/force_sp_Y
//     PlcTask Inputs/MAIN.force_sp_Z[129] <-> Status process data mapping/force_sp_Z
//     PlcTask Inputs/MAIN.pwm1[129] <-> Status process data mapping/pwm1
//     PlcTask Inputs/MAIN.pwm2[129] <-> Status process data mapping/pwm2
//     PlcTask Inputs/MAIN.pwm3[129] <-> Status process data mapping/pwm3
//     PlcTask Outputs/MAIN.enable_cmd[129] <-> Control process data mapping/enable
//     PlcTask Outputs/MAIN.force_cmd_X[129] <-> Control process data mapping/force_sp_X
//     PlcTask Outputs/MAIN.force_cmd_Y[129] <-> Control process data mapping/force_sp_Y
//     PlcTask Outputs/MAIN.force_cmd_Z[129] <-> Control process data mapping/force_sp_Z
//     PlcTask Outputs/MAIN.msthb[138] <-> Control process data mapping/msthb
//   SAsetGains/SAsetGains Instance <-> Device 1 (EtherCAT)/Box 131 (m1eph)/Box 139 (m1sa)
//     PlcTask Inputs/MAIN.cloop_stat[130] <-> Status process data mapping/close_loop
//     PlcTask Inputs/MAIN.enable_stat[130] <-> Status process data mapping/enable
//     PlcTask Inputs/MAIN.force_rb_X[130] <-> Status process data mapping/force_rb_X
//     PlcTask Inputs/MAIN.force_rb_Y[130] <-> Status process data mapping/force_rb_Y
//     PlcTask Inputs/MAIN.force_rb_Z[130] <-> Status process data mapping/force_rb_Z
//     PlcTask Inputs/MAIN.force_sp_X[130] <-> Status process data mapping/force_sp_X
//     PlcTask Inputs/MAIN.force_sp_Y[130] <-> Status process data mapping/force_sp_Y
//     PlcTask Inputs/MAIN.force_sp_Z[130] <-> Status process data mapping/force_sp_Z
//     PlcTask Inputs/MAIN.pwm1[130] <-> Status process data mapping/pwm1
//     PlcTask Inputs/MAIN.pwm2[130] <-> Status process data mapping/pwm2
//     PlcTask Inputs/MAIN.pwm3[130] <-> Status process data mapping/pwm3
//     PlcTask Outputs/MAIN.enable_cmd[130] <-> Control process data mapping/enable
//     PlcTask Outputs/MAIN.force_cmd_X[130] <-> Control process data mapping/force_sp_X
//     PlcTask Outputs/MAIN.force_cmd_Y[130] <-> Control process data mapping/force_sp_Y
//     PlcTask Outputs/MAIN.force_cmd_Z[130] <-> Control process data mapping/force_sp_Z
//     PlcTask Outputs/MAIN.msthb[139] <-> Control process data mapping/msthb
//   SAsetGains/SAsetGains Instance <-> Device 1 (EtherCAT)/Box 131 (m1eph)/Box 140 (m1sa)
//     PlcTask Inputs/MAIN.cloop_stat[131] <-> Status process data mapping/close_loop
//     PlcTask Inputs/MAIN.enable_stat[131] <-> Status process data mapping/enable
//     PlcTask Inputs/MAIN.force_rb_X[131] <-> Status process data mapping/force_rb_X
//     PlcTask Inputs/MAIN.force_rb_Y[131] <-> Status process data mapping/force_rb_Y
//     PlcTask Inputs/MAIN.force_rb_Z[131] <-> Status process data mapping/force_rb_Z
//     PlcTask Inputs/MAIN.force_sp_X[131] <-> Status process data mapping/force_sp_X
//     PlcTask Inputs/MAIN.force_sp_Y[131] <-> Status process data mapping/force_sp_Y
//     PlcTask Inputs/MAIN.force_sp_Z[131] <-> Status process data mapping/force_sp_Z
//     PlcTask Inputs/MAIN.pwm1[131] <-> Status process data mapping/pwm1
//     PlcTask Inputs/MAIN.pwm2[131] <-> Status process data mapping/pwm2
//     PlcTask Inputs/MAIN.pwm3[131] <-> Status process data mapping/pwm3
//     PlcTask Outputs/MAIN.enable_cmd[131] <-> Control process data mapping/enable
//     PlcTask Outputs/MAIN.force_cmd_X[131] <-> Control process data mapping/force_sp_X
//     PlcTask Outputs/MAIN.force_cmd_Y[131] <-> Control process data mapping/force_sp_Y
//     PlcTask Outputs/MAIN.force_cmd_Z[131] <-> Control process data mapping/force_sp_Z
//     PlcTask Outputs/MAIN.msthb[140] <-> Control process data mapping/msthb
//   SAsetGains/SAsetGains Instance <-> Device 1 (EtherCAT)/Box 131 (m1eph)/Box 141 (m1sa)
//     PlcTask Inputs/MAIN.cloop_stat[132] <-> Status process data mapping/close_loop
//     PlcTask Inputs/MAIN.enable_stat[132] <-> Status process data mapping/enable
//     PlcTask Inputs/MAIN.force_rb_X[132] <-> Status process data mapping/force_rb_X
//     PlcTask Inputs/MAIN.force_rb_Y[132] <-> Status process data mapping/force_rb_Y
//     PlcTask Inputs/MAIN.force_rb_Z[132] <-> Status process data mapping/force_rb_Z
//     PlcTask Inputs/MAIN.force_sp_X[132] <-> Status process data mapping/force_sp_X
//     PlcTask Inputs/MAIN.force_sp_Y[132] <-> Status process data mapping/force_sp_Y
//     PlcTask Inputs/MAIN.force_sp_Z[132] <-> Status process data mapping/force_sp_Z
//     PlcTask Inputs/MAIN.pwm1[132] <-> Status process data mapping/pwm1
//     PlcTask Inputs/MAIN.pwm2[132] <-> Status process data mapping/pwm2
//     PlcTask Inputs/MAIN.pwm3[132] <-> Status process data mapping/pwm3
//     PlcTask Outputs/MAIN.enable_cmd[132] <-> Control process data mapping/enable
//     PlcTask Outputs/MAIN.force_cmd_X[132] <-> Control process data mapping/force_sp_X
//     PlcTask Outputs/MAIN.force_cmd_Y[132] <-> Control process data mapping/force_sp_Y
//     PlcTask Outputs/MAIN.force_cmd_Z[132] <-> Control process data mapping/force_sp_Z
//     PlcTask Outputs/MAIN.msthb[141] <-> Control process data mapping/msthb
//   SAsetGains/SAsetGains Instance <-> Device 1 (EtherCAT)/Box 131 (m1eph)/Box 142 (m1sa)
//     PlcTask Inputs/MAIN.cloop_stat[133] <-> Status process data mapping/close_loop
//     PlcTask Inputs/MAIN.enable_stat[133] <-> Status process data mapping/enable
//     PlcTask Inputs/MAIN.force_rb_X[133] <-> Status process data mapping/force_rb_X
//     PlcTask Inputs/MAIN.force_rb_Y[133] <-> Status process data mapping/force_rb_Y
//     PlcTask Inputs/MAIN.force_rb_Z[133] <-> Status process data mapping/force_rb_Z
//     PlcTask Inputs/MAIN.force_sp_X[133] <-> Status process data mapping/force_sp_X
//     PlcTask Inputs/MAIN.force_sp_Y[133] <-> Status process data mapping/force_sp_Y
//     PlcTask Inputs/MAIN.force_sp_Z[133] <-> Status process data mapping/force_sp_Z
//     PlcTask Inputs/MAIN.pwm1[133] <-> Status process data mapping/pwm1
//     PlcTask Inputs/MAIN.pwm2[133] <-> Status process data mapping/pwm2
//     PlcTask Inputs/MAIN.pwm3[133] <-> Status process data mapping/pwm3
//     PlcTask Outputs/MAIN.enable_cmd[133] <-> Control process data mapping/enable
//     PlcTask Outputs/MAIN.force_cmd_X[133] <-> Control process data mapping/force_sp_X
//     PlcTask Outputs/MAIN.force_cmd_Y[133] <-> Control process data mapping/force_sp_Y
//     PlcTask Outputs/MAIN.force_cmd_Z[133] <-> Control process data mapping/force_sp_Z
//     PlcTask Outputs/MAIN.msthb[142] <-> Control process data mapping/msthb
//   SAsetGains/SAsetGains Instance <-> Device 1 (EtherCAT)/Box 131 (m1eph)/Box 143 (m1sa)
//     PlcTask Inputs/MAIN.cloop_stat[134] <-> Status process data mapping/close_loop
//     PlcTask Inputs/MAIN.enable_stat[134] <-> Status process data mapping/enable
//     PlcTask Inputs/MAIN.force_rb_X[134] <-> Status process data mapping/force_rb_X
//     PlcTask Inputs/MAIN.force_rb_Y[134] <-> Status process data mapping/force_rb_Y
//     PlcTask Inputs/MAIN.force_rb_Z[134] <-> Status process data mapping/force_rb_Z
//     PlcTask Inputs/MAIN.force_sp_X[134] <-> Status process data mapping/force_sp_X
//     PlcTask Inputs/MAIN.force_sp_Y[134] <-> Status process data mapping/force_sp_Y
//     PlcTask Inputs/MAIN.force_sp_Z[134] <-> Status process data mapping/force_sp_Z
//     PlcTask Inputs/MAIN.pwm1[134] <-> Status process data mapping/pwm1
//     PlcTask Inputs/MAIN.pwm2[134] <-> Status process data mapping/pwm2
//     PlcTask Inputs/MAIN.pwm3[134] <-> Status process data mapping/pwm3
//     PlcTask Outputs/MAIN.enable_cmd[134] <-> Control process data mapping/enable
//     PlcTask Outputs/MAIN.force_cmd_X[134] <-> Control process data mapping/force_sp_X
//     PlcTask Outputs/MAIN.force_cmd_Y[134] <-> Control process data mapping/force_sp_Y
//     PlcTask Outputs/MAIN.force_cmd_Z[134] <-> Control process data mapping/force_sp_Z
//     PlcTask Outputs/MAIN.msthb[143] <-> Control process data mapping/msthb
//   SAsetGains/SAsetGains Instance <-> Device 1 (EtherCAT)/Box 131 (m1eph)/Box 144 (m1sa)
//     PlcTask Inputs/MAIN.cloop_stat[135] <-> Status process data mapping/close_loop
//     PlcTask Inputs/MAIN.enable_stat[135] <-> Status process data mapping/enable
//     PlcTask Inputs/MAIN.force_rb_X[135] <-> Status process data mapping/force_rb_X
//     PlcTask Inputs/MAIN.force_rb_Y[135] <-> Status process data mapping/force_rb_Y
//     PlcTask Inputs/MAIN.force_rb_Z[135] <-> Status process data mapping/force_rb_Z
//     PlcTask Inputs/MAIN.force_sp_X[135] <-> Status process data mapping/force_sp_X
//     PlcTask Inputs/MAIN.force_sp_Y[135] <-> Status process data mapping/force_sp_Y
//     PlcTask Inputs/MAIN.force_sp_Z[135] <-> Status process data mapping/force_sp_Z
//     PlcTask Inputs/MAIN.pwm1[135] <-> Status process data mapping/pwm1
//     PlcTask Inputs/MAIN.pwm2[135] <-> Status process data mapping/pwm2
//     PlcTask Inputs/MAIN.pwm3[135] <-> Status process data mapping/pwm3
//     PlcTask Outputs/MAIN.enable_cmd[135] <-> Control process data mapping/enable
//     PlcTask Outputs/MAIN.force_cmd_X[135] <-> Control process data mapping/force_sp_X
//     PlcTask Outputs/MAIN.force_cmd_Y[135] <-> Control process data mapping/force_sp_Y
//     PlcTask Outputs/MAIN.force_cmd_Z[135] <-> Control process data mapping/force_sp_Z
//     PlcTask Outputs/MAIN.msthb[144] <-> Control process data mapping/msthb
//   SAsetGains/SAsetGains Instance <-> Device 1 (EtherCAT)/Box 131 (m1eph)/Box 145 (m1sa)
//     PlcTask Inputs/MAIN.cloop_stat[136] <-> Status process data mapping/close_loop
//     PlcTask Inputs/MAIN.enable_stat[136] <-> Status process data mapping/enable
//     PlcTask Inputs/MAIN.force_rb_X[136] <-> Status process data mapping/force_rb_X
//     PlcTask Inputs/MAIN.force_rb_Y[136] <-> Status process data mapping/force_rb_Y
//     PlcTask Inputs/MAIN.force_rb_Z[136] <-> Status process data mapping/force_rb_Z
//     PlcTask Inputs/MAIN.force_sp_X[136] <-> Status process data mapping/force_sp_X
//     PlcTask Inputs/MAIN.force_sp_Y[136] <-> Status process data mapping/force_sp_Y
//     PlcTask Inputs/MAIN.force_sp_Z[136] <-> Status process data mapping/force_sp_Z
//     PlcTask Inputs/MAIN.pwm1[136] <-> Status process data mapping/pwm1
//     PlcTask Inputs/MAIN.pwm2[136] <-> Status process data mapping/pwm2
//     PlcTask Inputs/MAIN.pwm3[136] <-> Status process data mapping/pwm3
//     PlcTask Outputs/MAIN.enable_cmd[136] <-> Control process data mapping/enable
//     PlcTask Outputs/MAIN.force_cmd_X[136] <-> Control process data mapping/force_sp_X
//     PlcTask Outputs/MAIN.force_cmd_Y[136] <-> Control process data mapping/force_sp_Y
//     PlcTask Outputs/MAIN.force_cmd_Z[136] <-> Control process data mapping/force_sp_Z
//     PlcTask Outputs/MAIN.msthb[145] <-> Control process data mapping/msthb
//   SAsetGains/SAsetGains Instance <-> Device 1 (EtherCAT)/Box 131 (m1eph)/Box 146 (m1sa)
//     PlcTask Inputs/MAIN.cloop_stat[137] <-> Status process data mapping/close_loop
//     PlcTask Inputs/MAIN.enable_stat[137] <-> Status process data mapping/enable
//     PlcTask Inputs/MAIN.force_rb_X[137] <-> Status process data mapping/force_rb_X
//     PlcTask Inputs/MAIN.force_rb_Y[137] <-> Status process data mapping/force_rb_Y
//     PlcTask Inputs/MAIN.force_rb_Z[137] <-> Status process data mapping/force_rb_Z
//     PlcTask Inputs/MAIN.force_sp_X[137] <-> Status process data mapping/force_sp_X
//     PlcTask Inputs/MAIN.force_sp_Y[137] <-> Status process data mapping/force_sp_Y
//     PlcTask Inputs/MAIN.force_sp_Z[137] <-> Status process data mapping/force_sp_Z
//     PlcTask Inputs/MAIN.pwm1[137] <-> Status process data mapping/pwm1
//     PlcTask Inputs/MAIN.pwm2[137] <-> Status process data mapping/pwm2
//     PlcTask Inputs/MAIN.pwm3[137] <-> Status process data mapping/pwm3
//     PlcTask Outputs/MAIN.enable_cmd[137] <-> Control process data mapping/enable
//     PlcTask Outputs/MAIN.force_cmd_X[137] <-> Control process data mapping/force_sp_X
//     PlcTask Outputs/MAIN.force_cmd_Y[137] <-> Control process data mapping/force_sp_Y
//     PlcTask Outputs/MAIN.force_cmd_Z[137] <-> Control process data mapping/force_sp_Z
//     PlcTask Outputs/MAIN.msthb[146] <-> Control process data mapping/msthb
//   SAsetGains/SAsetGains Instance <-> Device 1 (EtherCAT)/Box 131 (m1eph)/Box 147 (m1sa)
//     PlcTask Inputs/MAIN.cloop_stat[138] <-> Status process data mapping/close_loop
//     PlcTask Inputs/MAIN.enable_stat[138] <-> Status process data mapping/enable
//     PlcTask Inputs/MAIN.force_rb_X[138] <-> Status process data mapping/force_rb_X
//     PlcTask Inputs/MAIN.force_rb_Y[138] <-> Status process data mapping/force_rb_Y
//     PlcTask Inputs/MAIN.force_rb_Z[138] <-> Status process data mapping/force_rb_Z
//     PlcTask Inputs/MAIN.force_sp_X[138] <-> Status process data mapping/force_sp_X
//     PlcTask Inputs/MAIN.force_sp_Y[138] <-> Status process data mapping/force_sp_Y
//     PlcTask Inputs/MAIN.force_sp_Z[138] <-> Status process data mapping/force_sp_Z
//     PlcTask Inputs/MAIN.pwm1[138] <-> Status process data mapping/pwm1
//     PlcTask Inputs/MAIN.pwm2[138] <-> Status process data mapping/pwm2
//     PlcTask Inputs/MAIN.pwm3[138] <-> Status process data mapping/pwm3
//     PlcTask Outputs/MAIN.enable_cmd[138] <-> Control process data mapping/enable
//     PlcTask Outputs/MAIN.force_cmd_X[138] <-> Control process data mapping/force_sp_X
//     PlcTask Outputs/MAIN.force_cmd_Y[138] <-> Control process data mapping/force_sp_Y
//     PlcTask Outputs/MAIN.force_cmd_Z[138] <-> Control process data mapping/force_sp_Z
//     PlcTask Outputs/MAIN.msthb[147] <-> Control process data mapping/msthb
//   SAsetGains/SAsetGains Instance <-> Device 1 (EtherCAT)/Box 148 (m1eph)
//     PlcTask Outputs/MAIN.msthb[148] <-> Control process data mapping/msthb
//   SAsetGains/SAsetGains Instance <-> Device 1 (EtherCAT)/Box 148 (m1eph)/Box 149 (m1sa)
//     PlcTask Inputs/MAIN.cloop_stat[139] <-> Status process data mapping/close_loop
//     PlcTask Inputs/MAIN.enable_stat[139] <-> Status process data mapping/enable
//     PlcTask Inputs/MAIN.force_rb_X[139] <-> Status process data mapping/force_rb_X
//     PlcTask Inputs/MAIN.force_rb_Y[139] <-> Status process data mapping/force_rb_Y
//     PlcTask Inputs/MAIN.force_rb_Z[139] <-> Status process data mapping/force_rb_Z
//     PlcTask Inputs/MAIN.force_sp_X[139] <-> Status process data mapping/force_sp_X
//     PlcTask Inputs/MAIN.force_sp_Y[139] <-> Status process data mapping/force_sp_Y
//     PlcTask Inputs/MAIN.force_sp_Z[139] <-> Status process data mapping/force_sp_Z
//     PlcTask Inputs/MAIN.pwm1[139] <-> Status process data mapping/pwm1
//     PlcTask Inputs/MAIN.pwm2[139] <-> Status process data mapping/pwm2
//     PlcTask Inputs/MAIN.pwm3[139] <-> Status process data mapping/pwm3
//     PlcTask Outputs/MAIN.enable_cmd[139] <-> Control process data mapping/enable
//     PlcTask Outputs/MAIN.force_cmd_X[139] <-> Control process data mapping/force_sp_X
//     PlcTask Outputs/MAIN.force_cmd_Y[139] <-> Control process data mapping/force_sp_Y
//     PlcTask Outputs/MAIN.force_cmd_Z[139] <-> Control process data mapping/force_sp_Z
//     PlcTask Outputs/MAIN.msthb[149] <-> Control process data mapping/msthb
//   SAsetGains/SAsetGains Instance <-> Device 1 (EtherCAT)/Box 148 (m1eph)/Box 150 (m1sa)
//     PlcTask Inputs/MAIN.cloop_stat[140] <-> Status process data mapping/close_loop
//     PlcTask Inputs/MAIN.enable_stat[140] <-> Status process data mapping/enable
//     PlcTask Inputs/MAIN.force_rb_X[140] <-> Status process data mapping/force_rb_X
//     PlcTask Inputs/MAIN.force_rb_Y[140] <-> Status process data mapping/force_rb_Y
//     PlcTask Inputs/MAIN.force_rb_Z[140] <-> Status process data mapping/force_rb_Z
//     PlcTask Inputs/MAIN.force_sp_X[140] <-> Status process data mapping/force_sp_X
//     PlcTask Inputs/MAIN.force_sp_Y[140] <-> Status process data mapping/force_sp_Y
//     PlcTask Inputs/MAIN.force_sp_Z[140] <-> Status process data mapping/force_sp_Z
//     PlcTask Inputs/MAIN.pwm1[140] <-> Status process data mapping/pwm1
//     PlcTask Inputs/MAIN.pwm2[140] <-> Status process data mapping/pwm2
//     PlcTask Inputs/MAIN.pwm3[140] <-> Status process data mapping/pwm3
//     PlcTask Outputs/MAIN.enable_cmd[140] <-> Control process data mapping/enable
//     PlcTask Outputs/MAIN.force_cmd_X[140] <-> Control process data mapping/force_sp_X
//     PlcTask Outputs/MAIN.force_cmd_Y[140] <-> Control process data mapping/force_sp_Y
//     PlcTask Outputs/MAIN.force_cmd_Z[140] <-> Control process data mapping/force_sp_Z
//     PlcTask Outputs/MAIN.msthb[150] <-> Control process data mapping/msthb
//   SAsetGains/SAsetGains Instance <-> Device 1 (EtherCAT)/Box 148 (m1eph)/Box 151 (m1sa)
//     PlcTask Inputs/MAIN.cloop_stat[141] <-> Status process data mapping/close_loop
//     PlcTask Inputs/MAIN.enable_stat[141] <-> Status process data mapping/enable
//     PlcTask Inputs/MAIN.force_rb_X[141] <-> Status process data mapping/force_rb_X
//     PlcTask Inputs/MAIN.force_rb_Y[141] <-> Status process data mapping/force_rb_Y
//     PlcTask Inputs/MAIN.force_rb_Z[141] <-> Status process data mapping/force_rb_Z
//     PlcTask Inputs/MAIN.force_sp_X[141] <-> Status process data mapping/force_sp_X
//     PlcTask Inputs/MAIN.force_sp_Y[141] <-> Status process data mapping/force_sp_Y
//     PlcTask Inputs/MAIN.force_sp_Z[141] <-> Status process data mapping/force_sp_Z
//     PlcTask Inputs/MAIN.pwm1[141] <-> Status process data mapping/pwm1
//     PlcTask Inputs/MAIN.pwm2[141] <-> Status process data mapping/pwm2
//     PlcTask Inputs/MAIN.pwm3[141] <-> Status process data mapping/pwm3
//     PlcTask Outputs/MAIN.enable_cmd[141] <-> Control process data mapping/enable
//     PlcTask Outputs/MAIN.force_cmd_X[141] <-> Control process data mapping/force_sp_X
//     PlcTask Outputs/MAIN.force_cmd_Y[141] <-> Control process data mapping/force_sp_Y
//     PlcTask Outputs/MAIN.force_cmd_Z[141] <-> Control process data mapping/force_sp_Z
//     PlcTask Outputs/MAIN.msthb[151] <-> Control process data mapping/msthb
//   SAsetGains/SAsetGains Instance <-> Device 1 (EtherCAT)/Box 148 (m1eph)/Box 152 (m1sa)
//     PlcTask Inputs/MAIN.cloop_stat[142] <-> Status process data mapping/close_loop
//     PlcTask Inputs/MAIN.enable_stat[142] <-> Status process data mapping/enable
//     PlcTask Inputs/MAIN.force_rb_X[142] <-> Status process data mapping/force_rb_X
//     PlcTask Inputs/MAIN.force_rb_Y[142] <-> Status process data mapping/force_rb_Y
//     PlcTask Inputs/MAIN.force_rb_Z[142] <-> Status process data mapping/force_rb_Z
//     PlcTask Inputs/MAIN.force_sp_X[142] <-> Status process data mapping/force_sp_X
//     PlcTask Inputs/MAIN.force_sp_Y[142] <-> Status process data mapping/force_sp_Y
//     PlcTask Inputs/MAIN.force_sp_Z[142] <-> Status process data mapping/force_sp_Z
//     PlcTask Inputs/MAIN.pwm1[142] <-> Status process data mapping/pwm1
//     PlcTask Inputs/MAIN.pwm2[142] <-> Status process data mapping/pwm2
//     PlcTask Inputs/MAIN.pwm3[142] <-> Status process data mapping/pwm3
//     PlcTask Outputs/MAIN.enable_cmd[142] <-> Control process data mapping/enable
//     PlcTask Outputs/MAIN.force_cmd_X[142] <-> Control process data mapping/force_sp_X
//     PlcTask Outputs/MAIN.force_cmd_Y[142] <-> Control process data mapping/force_sp_Y
//     PlcTask Outputs/MAIN.force_cmd_Z[142] <-> Control process data mapping/force_sp_Z
//     PlcTask Outputs/MAIN.msthb[152] <-> Control process data mapping/msthb
//   SAsetGains/SAsetGains Instance <-> Device 1 (EtherCAT)/Box 148 (m1eph)/Box 153 (m1sa)
//     PlcTask Inputs/MAIN.cloop_stat[143] <-> Status process data mapping/close_loop
//     PlcTask Inputs/MAIN.enable_stat[143] <-> Status process data mapping/enable
//     PlcTask Inputs/MAIN.force_rb_X[143] <-> Status process data mapping/force_rb_X
//     PlcTask Inputs/MAIN.force_rb_Y[143] <-> Status process data mapping/force_rb_Y
//     PlcTask Inputs/MAIN.force_rb_Z[143] <-> Status process data mapping/force_rb_Z
//     PlcTask Inputs/MAIN.force_sp_X[143] <-> Status process data mapping/force_sp_X
//     PlcTask Inputs/MAIN.force_sp_Y[143] <-> Status process data mapping/force_sp_Y
//     PlcTask Inputs/MAIN.force_sp_Z[143] <-> Status process data mapping/force_sp_Z
//     PlcTask Inputs/MAIN.pwm1[143] <-> Status process data mapping/pwm1
//     PlcTask Inputs/MAIN.pwm2[143] <-> Status process data mapping/pwm2
//     PlcTask Inputs/MAIN.pwm3[143] <-> Status process data mapping/pwm3
//     PlcTask Outputs/MAIN.enable_cmd[143] <-> Control process data mapping/enable
//     PlcTask Outputs/MAIN.force_cmd_X[143] <-> Control process data mapping/force_sp_X
//     PlcTask Outputs/MAIN.force_cmd_Y[143] <-> Control process data mapping/force_sp_Y
//     PlcTask Outputs/MAIN.force_cmd_Z[143] <-> Control process data mapping/force_sp_Z
//     PlcTask Outputs/MAIN.msthb[153] <-> Control process data mapping/msthb
//   SAsetGains/SAsetGains Instance <-> Device 1 (EtherCAT)/Box 148 (m1eph)/Box 154 (m1sa)
//     PlcTask Inputs/MAIN.cloop_stat[144] <-> Status process data mapping/close_loop
//     PlcTask Inputs/MAIN.enable_stat[144] <-> Status process data mapping/enable
//     PlcTask Inputs/MAIN.force_rb_X[144] <-> Status process data mapping/force_rb_X
//     PlcTask Inputs/MAIN.force_rb_Y[144] <-> Status process data mapping/force_rb_Y
//     PlcTask Inputs/MAIN.force_rb_Z[144] <-> Status process data mapping/force_rb_Z
//     PlcTask Inputs/MAIN.force_sp_X[144] <-> Status process data mapping/force_sp_X
//     PlcTask Inputs/MAIN.force_sp_Y[144] <-> Status process data mapping/force_sp_Y
//     PlcTask Inputs/MAIN.force_sp_Z[144] <-> Status process data mapping/force_sp_Z
//     PlcTask Inputs/MAIN.pwm1[144] <-> Status process data mapping/pwm1
//     PlcTask Inputs/MAIN.pwm2[144] <-> Status process data mapping/pwm2
//     PlcTask Inputs/MAIN.pwm3[144] <-> Status process data mapping/pwm3
//     PlcTask Outputs/MAIN.enable_cmd[144] <-> Control process data mapping/enable
//     PlcTask Outputs/MAIN.force_cmd_X[144] <-> Control process data mapping/force_sp_X
//     PlcTask Outputs/MAIN.force_cmd_Y[144] <-> Control process data mapping/force_sp_Y
//     PlcTask Outputs/MAIN.force_cmd_Z[144] <-> Control process data mapping/force_sp_Z
//     PlcTask Outputs/MAIN.msthb[154] <-> Control process data mapping/msthb
//   SAsetGains/SAsetGains Instance <-> Device 1 (EtherCAT)/Box 148 (m1eph)/Box 155 (m1sa)
//     PlcTask Inputs/MAIN.cloop_stat[145] <-> Status process data mapping/close_loop
//     PlcTask Inputs/MAIN.enable_stat[145] <-> Status process data mapping/enable
//     PlcTask Inputs/MAIN.force_rb_X[145] <-> Status process data mapping/force_rb_X
//     PlcTask Inputs/MAIN.force_rb_Y[145] <-> Status process data mapping/force_rb_Y
//     PlcTask Inputs/MAIN.force_rb_Z[145] <-> Status process data mapping/force_rb_Z
//     PlcTask Inputs/MAIN.force_sp_X[145] <-> Status process data mapping/force_sp_X
//     PlcTask Inputs/MAIN.force_sp_Y[145] <-> Status process data mapping/force_sp_Y
//     PlcTask Inputs/MAIN.force_sp_Z[145] <-> Status process data mapping/force_sp_Z
//     PlcTask Inputs/MAIN.pwm1[145] <-> Status process data mapping/pwm1
//     PlcTask Inputs/MAIN.pwm2[145] <-> Status process data mapping/pwm2
//     PlcTask Inputs/MAIN.pwm3[145] <-> Status process data mapping/pwm3
//     PlcTask Outputs/MAIN.enable_cmd[145] <-> Control process data mapping/enable
//     PlcTask Outputs/MAIN.force_cmd_X[145] <-> Control process data mapping/force_sp_X
//     PlcTask Outputs/MAIN.force_cmd_Y[145] <-> Control process data mapping/force_sp_Y
//     PlcTask Outputs/MAIN.force_cmd_Z[145] <-> Control process data mapping/force_sp_Z
//     PlcTask Outputs/MAIN.msthb[155] <-> Control process data mapping/msthb
//   SAsetGains/SAsetGains Instance <-> Device 1 (EtherCAT)/Box 148 (m1eph)/Box 156 (m1sa)
//     PlcTask Inputs/MAIN.cloop_stat[146] <-> Status process data mapping/close_loop
//     PlcTask Inputs/MAIN.enable_stat[146] <-> Status process data mapping/enable
